LIN {X 0.029,Y -222.259,Z 1297.820,A 0.000,B 0.000,C 90.000,E1 327.533} C_DIS
LIN {X -0.001,Y -229.136,Z 1297.798,A 0.000,B 0.000,C 90.000,E1 323.703} C_DIS
LIN {X 0.049,Y -236.925,Z 1297.777,A 0.000,B 0.000,C 90.000,E1 319.908} C_DIS
LIN {X -0.024,Y -243.959,Z 1297.761,A 0.000,B 0.000,C 90.000,E1 316.944} C_DIS
LIN {X 0.067,Y -252.924,Z 1297.742,A 0.000,B 0.000,C 90.000,E1 313.623} C_DIS
LIN {X -0.154,Y -260.714,Z 1297.728,A 0.000,B 0.000,C 90.000,E1 311.148} C_DIS
LIN {X -0.101,Y -267.095,Z 1297.719,A 0.000,B 0.000,C 90.000,E1 309.358} C_DIS
LIN {X -0.026,Y -275.499,Z 1297.707,A 0.000,B 0.000,C 90.000,E1 307.237} C_DIS
LIN {X -0.075,Y -283.266,Z 1297.697,A 0.000,B 0.000,C 90.000,E1 305.518} C_DIS
LIN {X 0.052,Y -293.703,Z 1297.686,A 0.000,B 0.000,C 90.000,E1 303.452} C_DIS
LIN {X -0.037,Y -303.212,Z 1297.677,A 0.000,B 0.000,C 90.000,E1 301.799} C_DIS
LIN {X 0.071,Y -318.318,Z 1297.664,A 0.000,B 0.000,C 90.000,E1 299.489} C_DIS
LIN {X 0.040,Y -330.289,Z 1297.655,A 0.000,B 0.000,C 90.000,E1 297.897} C_DIS
LIN {X 0.050,Y -350.836,Z 1297.641,A 0.000,B 0.000,C 90.000,E1 295.412} C_DIS
LIN {X 0.152,Y -363.810,Z 1297.633,A 0.000,B 0.000,C 90.000,E1 293.898} C_DIS
LIN {X -0.055,Y -376.466,Z 1297.625,A 0.000,B 0.000,C 90.000,E1 292.461} C_DIS
LIN {X 0.202,Y -388.826,Z 1297.617,A 0.000,B 0.000,C 90.000,E1 290.972} C_DIS
LIN {X 0.126,Y -413.426,Z 1297.601,A 0.000,B 0.000,C 90.000,E1 288.181} C_DIS
LIN {X -0.186,Y -425.633,Z 1297.594,A 0.000,B 0.000,C 90.000,E1 286.858} C_DIS
LIN {X 0.004,Y -432.572,Z 1297.589,A 0.000,B 0.000,C 90.000,E1 286.024} C_DIS
LIN {X -0.170,Y -438.889,Z 1297.585,A 0.000,B 0.000,C 90.000,E1 285.245} C_DIS
LIN {X -0.194,Y -442.664,Z 1297.582,A 0.000,B 0.000,C 90.000,E1 284.717} C_DIS
LIN {X 0.140,Y -447.628,Z 1297.577,A 0.000,B 0.000,C 90.000,E1 283.883} C_DIS
LIN {X -0.016,Y -451.995,Z 1297.573,A 0.000,B 0.000,C 90.000,E1 283.119} C_DIS
LIN {X -0.140,Y -455.836,Z 1297.568,A 0.000,B 0.000,C 90.000,E1 282.355} C_DIS
LIN {X -0.055,Y -458.106,Z 1297.566,A 0.000,B 0.000,C 90.000,E1 281.827} C_DIS
LIN {X 0.044,Y -460.116,Z 1297.563,A 0.000,B 0.000,C 90.000,E1 281.299} C_DIS
LIN {X 0.063,Y -461.853,Z 1297.560,A 0.000,B 0.000,C 90.000,E1 280.782} C_DIS
LIN {X 0.181,Y -463.242,Z 1297.557,A 0.000,B 0.000,C 90.000,E1 280.254} C_DIS
LIN {X -0.150,Y -464.264,Z 1297.554,A 0.000,B 0.000,C 90.000,E1 279.782} C_DIS
LIN {X -0.095,Y -464.907,Z 1297.551,A 0.000,B 0.000,C 90.000,E1 279.265} C_DIS
LIN {X -0.030,Y -465.112,Z 1297.549,A 0.000,B 0.000,C 90.000,E1 278.746} C_DIS
LIN {X 0.108,Y -464.850,Z 1297.546,A 0.000,B 0.000,C 90.000,E1 278.219} C_DIS
LIN {X 0.179,Y -464.126,Z 1297.543,A 0.000,B 0.000,C 90.000,E1 277.701} C_DIS
LIN {X -0.210,Y -462.917,Z 1297.540,A 0.000,B 0.000,C 90.000,E1 277.239} C_DIS
LIN {X -0.142,Y -461.245,Z 1297.537,A 0.000,B 0.000,C 90.000,E1 276.720} C_DIS
LIN {X -0.081,Y -459.120,Z 1297.534,A 0.000,B 0.000,C 90.000,E1 276.201} C_DIS
LIN {X -0.030,Y -456.577,Z 1297.531,A 0.000,B 0.000,C 90.000,E1 275.682} C_DIS
LIN {X 0.001,Y -453.548,Z 1297.529,A 0.000,B 0.000,C 90.000,E1 275.163} C_DIS
LIN {X 0.013,Y -449.938,Z 1297.526,A 0.000,B 0.000,C 90.000,E1 274.645} C_DIS
LIN {X -0.028,Y -445.480,Z 1297.523,A 0.000,B 0.000,C 90.000,E1 274.131} C_DIS
LIN {X 0.194,Y -442.859,Z 1297.521,A 0.000,B 0.000,C 90.000,E1 273.841} C_DIS
LIN {X -0.088,Y -437.026,Z 1297.519,A 0.000,B 0.000,C 90.000,E1 273.383} C_DIS
LIN {X 0.058,Y -430.812,Z 1297.516,A 0.000,B 0.000,C 90.000,E1 272.922} C_DIS
LIN {X 0.169,Y -424.141,Z 1297.514,A 0.000,B 0.000,C 90.000,E1 272.522} C_DIS
LIN {X -0.134,Y -417.304,Z 1297.512,A 0.000,B 0.000,C 90.000,E1 272.236} C_DIS
LIN {X -0.049,Y -410.193,Z 1297.511,A 0.000,B 0.000,C 90.000,E1 271.949} C_DIS
LIN {X -0.028,Y -403.093,Z 1297.510,A 0.000,B 0.000,C 90.000,E1 271.718} C_DIS
LIN {X -0.139,Y -395.840,Z 1297.508,A 0.000,B 0.000,C 90.000,E1 271.547} C_DIS
LIN {X -0.014,Y -388.314,Z 1297.508,A 0.000,B 0.000,C 90.000,E1 271.375} C_DIS
LIN {X -0.082,Y -379.859,Z 1297.507,A 0.000,B 0.000,C 90.000,E1 271.260} C_DIS
LIN {X 0.025,Y -369.869,Z 1297.506,A 0.000,B 0.000,C 90.000,E1 271.146} C_DIS
LIN {X 0.116,Y -361.500,Z 1297.506,A 0.000,B 0.000,C 90.000,E1 271.088} C_DIS
LIN {X 0.020,Y -355.047,Z 1297.506,A 0.000,B 0.000,C 90.000,E1 271.088} C_DIS
LIN {X -0.014,Y -181.437,Z 1297.506,A 0.000,B 0.000,C 90.000,E1 271.088} C_DIS
LIN {X -0.077,Y -181.580,Z 1297.501,A 0.000,B 0.000,C 90.000,E1 270.229} C_DIS
LIN {X 0.092,Y -180.889,Z 1297.473,A 0.000,B 0.000,C 90.000,E1 265.122} C_DIS
LIN {X -0.026,Y -179.014,Z 1297.445,A 0.000,B 0.000,C 90.000,E1 260.095} C_DIS
LIN {X 0.069,Y -178.636,Z 1297.440,A 0.000,B 0.000,C 90.000,E1 259.218} C_DIS
LIN {X -0.033,Y -175.686,Z 1297.412,A 0.000,B 0.000,C 90.000,E1 254.157} C_DIS
LIN {X -0.022,Y -172.403,Z 1297.388,A 0.000,B 0.000,C 90.000,E1 249.880} C_DIS
LIN {X -0.005,Y -171.214,Z 1297.379,A 0.000,B 0.000,C 90.000,E1 248.156} C_DIS
LIN {X -0.029,Y -167.498,Z 1297.355,A 0.000,B 0.000,C 90.000,E1 243.845} C_DIS
LIN {X 0.053,Y -166.894,Z 1297.350,A 0.000,B 0.000,C 90.000,E1 242.948} C_DIS
LIN {X 0.043,Y -162.201,Z 1297.321,A 0.000,B 0.000,C 90.000,E1 237.709} C_DIS
LIN {X 0.011,Y -160.774,Z 1297.311,A 0.000,B 0.000,C 90.000,E1 235.960} C_DIS
LIN {X -0.018,Y -157.568,Z 1297.291,A 0.000,B 0.000,C 90.000,E1 232.431} C_DIS
LIN {X 0.017,Y -155.599,Z 1297.276,A 0.000,B 0.000,C 90.000,E1 229.747} C_DIS
LIN {X 0.067,Y -151.880,Z 1297.251,A 0.000,B 0.000,C 90.000,E1 225.243} C_DIS
LIN {X 0.081,Y -150.106,Z 1297.236,A 0.000,B 0.000,C 90.000,E1 222.528} C_DIS
LIN {X -0.003,Y -146.903,Z 1297.211,A 0.000,B 0.000,C 90.000,E1 218.016} C_DIS
LIN {X 0.017,Y -145.490,Z 1297.196,A 0.000,B 0.000,C 90.000,E1 215.264} C_DIS
LIN {X 0.017,Y -142.897,Z 1297.170,A 0.000,B 0.000,C 90.000,E1 210.669} C_DIS
LIN {X -0.052,Y -141.516,Z 1297.150,A 0.000,B 0.000,C 90.000,E1 207.001} C_DIS
LIN {X -0.009,Y -139.393,Z 1297.114,A 0.000,B 0.000,C 90.000,E1 200.482} C_DIS
LIN {X 0.042,Y -139.104,Z 1297.103,A 0.000,B 0.000,C 90.000,E1 198.598} C_DIS
LIN {X 0.034,Y -138.353,Z 1297.057,A 0.000,B 0.000,C 90.000,E1 190.197} C_DIS
LIN {X 0.027,Y -139.512,Z 1297.005,A 0.000,B 0.000,C 90.000,E1 180.859} C_DIS
LIN {X -0.032,Y -141.159,Z 1296.974,A 0.000,B 0.000,C 90.000,E1 175.298} C_DIS
LIN {X -0.061,Y -142.539,Z 1296.958,A 0.000,B 0.000,C 90.000,E1 172.527} C_DIS
LIN {X 0.006,Y -144.809,Z 1296.933,A 0.000,B 0.000,C 90.000,E1 167.881} C_DIS
LIN {X -0.006,Y -147.428,Z 1296.912,A 0.000,B 0.000,C 90.000,E1 164.212} C_DIS
LIN {X 0.022,Y -150.008,Z 1296.892,A 0.000,B 0.000,C 90.000,E1 160.550} C_DIS
LIN {X 0.030,Y -153.339,Z 1296.872,A 0.000,B 0.000,C 90.000,E1 156.922} C_DIS
LIN {X 0.011,Y -155.874,Z 1296.857,A 0.000,B 0.000,C 90.000,E1 154.229} C_DIS
LIN {X -0.022,Y -159.728,Z 1296.837,A 0.000,B 0.000,C 90.000,E1 150.667} C_DIS
LIN {X 0.044,Y -161.967,Z 1296.827,A 0.000,B 0.000,C 90.000,E1 148.869} C_DIS
LIN {X -0.071,Y -166.158,Z 1296.808,A 0.000,B 0.000,C 90.000,E1 145.388} C_DIS
LIN {X -0.076,Y -171.172,Z 1296.788,A 0.000,B 0.000,C 90.000,E1 141.904} C_DIS
LIN {X -0.042,Y -176.052,Z 1296.769,A 0.000,B 0.000,C 90.000,E1 138.447} C_DIS
LIN {X -0.047,Y -180.308,Z 1296.755,A 0.000,B 0.000,C 90.000,E1 135.891} C_DIS
LIN {X -0.076,Y -185.719,Z 1296.736,A 0.000,B 0.000,C 90.000,E1 132.528} C_DIS
LIN {X -0.024,Y -190.327,Z 1296.722,A 0.000,B 0.000,C 90.000,E1 130.011} C_DIS
LIN {X 0.023,Y -197.653,Z 1296.699,A 0.000,B 0.000,C 90.000,E1 125.884} C_DIS
LIN {X -0.040,Y -199.574,Z 1296.694,A 0.000,B 0.000,C 90.000,E1 124.945} C_DIS
LIN {X -0.098,Y -309.336,Z 1296.694,A 0.000,B 0.000,C 90.000,E1 124.945} C_DIS
LIN {X -0.078,Y -311.539,Z 1296.694,A 0.000,B 0.000,C 90.000,E1 124.898} C_DIS
LIN {X 0.053,Y -316.988,Z 1296.692,A 0.000,B 0.000,C 90.000,E1 124.565} C_DIS
LIN {X -0.076,Y -319.924,Z 1296.690,A 0.000,B 0.000,C 90.000,E1 124.278} C_DIS
LIN {X -0.103,Y -321.931,Z 1296.689,A 0.000,B 0.000,C 90.000,E1 123.992} C_DIS
LIN {X -0.130,Y -323.499,Z 1296.687,A 0.000,B 0.000,C 90.000,E1 123.706} C_DIS
LIN {X -0.043,Y -324.854,Z 1296.685,A 0.000,B 0.000,C 90.000,E1 123.372} C_DIS
LIN {X 0.054,Y -336.500,Z 1296.668,A 0.000,B 0.000,C 90.000,E1 120.207} C_DIS
LIN {X 0.008,Y -348.385,Z 1296.652,A 0.000,B 0.000,C 90.000,E1 117.436} C_DIS
LIN {X -0.025,Y -361.721,Z 1296.637,A 0.000,B 0.000,C 90.000,E1 114.719} C_DIS
LIN {X 0.081,Y -374.891,Z 1296.624,A 0.000,B 0.000,C 90.000,E1 112.333} C_DIS
LIN {X 0.233,Y -389.393,Z 1296.611,A 0.000,B 0.000,C 90.000,E1 109.993} C_DIS
LIN {X -0.019,Y -405.329,Z 1296.599,A 0.000,B 0.000,C 90.000,E1 107.764} C_DIS
LIN {X 0.002,Y -422.809,Z 1296.586,A 0.000,B 0.000,C 90.000,E1 105.552} C_DIS
LIN {X -0.060,Y -441.930,Z 1296.574,A 0.000,B 0.000,C 90.000,E1 103.411} C_DIS
LIN {X -0.233,Y -462.017,Z 1296.563,A 0.000,B 0.000,C 90.000,E1 101.422} C_DIS
LIN {X -0.198,Y -477.377,Z 1296.556,A 0.000,B 0.000,C 90.000,E1 100.018} C_DIS
LIN {X -0.117,Y -479.361,Z 1296.554,A 0.000,B 0.000,C 90.000,E1 99.782} C_DIS
LIN {X 0.148,Y -481.022,Z 1296.553,A 0.000,B 0.000,C 90.000,E1 99.500} C_DIS
LIN {X 0.022,Y -482.268,Z 1296.552,A 0.000,B 0.000,C 90.000,E1 99.265} C_DIS
LIN {X 0.188,Y -483.795,Z 1296.549,A 0.000,B 0.000,C 90.000,E1 98.746} C_DIS
LIN {X -0.046,Y -484.267,Z 1296.546,A 0.000,B 0.000,C 90.000,E1 98.276} C_DIS
LIN {X 0.136,Y -483.763,Z 1296.543,A 0.000,B 0.000,C 90.000,E1 97.757} C_DIS
LIN {X -0.156,Y -482.204,Z 1296.540,A 0.000,B 0.000,C 90.000,E1 97.296} C_DIS
LIN {X 0.145,Y -480.944,Z 1296.539,A 0.000,B 0.000,C 90.000,E1 97.011} C_DIS
LIN {X 0.028,Y -479.266,Z 1296.538,A 0.000,B 0.000,C 90.000,E1 96.777} C_DIS
LIN {X -0.011,Y -467.993,Z 1296.529,A 0.000,B 0.000,C 90.000,E1 95.277} C_DIS
LIN {X 0.186,Y -454.112,Z 1296.518,A 0.000,B 0.000,C 90.000,E1 93.212} C_DIS
LIN {X -0.019,Y -437.481,Z 1296.504,A 0.000,B 0.000,C 90.000,E1 90.630} C_DIS
LIN {X -0.017,Y -419.690,Z 1296.486,A 0.000,B 0.000,C 90.000,E1 87.421} C_DIS
LIN {X -0.061,Y -408.148,Z 1296.474,A 0.000,B 0.000,C 90.000,E1 85.241} C_DIS
LIN {X 0.054,Y -397.889,Z 1296.463,A 0.000,B 0.000,C 90.000,E1 83.280} C_DIS
LIN {X -0.039,Y -387.490,Z 1296.452,A 0.000,B 0.000,C 90.000,E1 81.319} C_DIS
LIN {X 0.115,Y -378.224,Z 1296.442,A 0.000,B 0.000,C 90.000,E1 79.577} C_DIS
LIN {X -0.197,Y -370.312,Z 1296.434,A 0.000,B 0.000,C 90.000,E1 78.173} C_DIS
LIN {X 0.150,Y -360.564,Z 1296.424,A 0.000,B 0.000,C 90.000,E1 76.353} C_DIS
LIN {X -0.012,Y -348.993,Z 1296.413,A 0.000,B 0.000,C 90.000,E1 74.283} C_DIS
LIN {X 0.100,Y -337.395,Z 1296.401,A 0.000,B 0.000,C 90.000,E1 72.127} C_DIS
LIN {X 0.029,Y -324.338,Z 1296.387,A 0.000,B 0.000,C 90.000,E1 69.645} C_DIS
LIN {X -0.165,Y -309.001,Z 1296.369,A 0.000,B 0.000,C 90.000,E1 66.485} C_DIS
LIN {X -0.029,Y -296.366,Z 1296.353,A 0.000,B 0.000,C 90.000,E1 63.512} C_DIS
LIN {X -0.050,Y -288.933,Z 1296.342,A 0.000,B 0.000,C 90.000,E1 61.513} C_DIS
LIN {X 0.010,Y -280.189,Z 1296.327,A 0.000,B 0.000,C 90.000,E1 58.791} C_DIS
LIN {X 0.034,Y -270.342,Z 1296.307,A 0.000,B 0.000,C 90.000,E1 55.341} C_DIS
LIN {X 0.075,Y -261.296,Z 1296.288,A 0.000,B 0.000,C 90.000,E1 51.823} C_DIS
LIN {X -0.107,Y -254.319,Z 1296.272,A 0.000,B 0.000,C 90.000,E1 49.013} C_DIS
LIN {X -0.150,Y -247.597,Z 1296.256,A 0.000,B 0.000,C 90.000,E1 46.134} C_DIS
LIN {X -0.057,Y -239.525,Z 1296.236,A 0.000,B 0.000,C 90.000,E1 42.447} C_DIS
LIN {X 0.013,Y -232.214,Z 1296.215,A 0.000,B 0.000,C 90.000,E1 38.705} C_DIS
LIN {X -0.069,Y -225.785,Z 1296.194,A 0.000,B 0.000,C 90.000,E1 34.945} C_DIS
LIN {X 0.062,Y -220.215,Z 1296.173,A 0.000,B 0.000,C 90.000,E1 31.082} C_DIS
LIN {X 0.070,Y -215.505,Z 1296.151,A 0.000,B 0.000,C 90.000,E1 27.206} C_DIS
LIN {X 0.045,Y -210.493,Z 1296.125,A 0.000,B 0.000,C 90.000,E1 22.514} C_DIS
LIN {X -0.087,Y -206.837,Z 1296.103,A 0.000,B 0.000,C 90.000,E1 18.598} C_DIS
LIN {X 0.065,Y -203.016,Z 1296.077,A 0.000,B 0.000,C 90.000,E1 13.772} C_DIS
LIN {X -0.013,Y -200.039,Z 1296.050,A 0.000,B 0.000,C 90.000,E1 8.973} C_DIS
LIN {X -0.086,Y -197.636,Z 1296.014,A 0.000,B 0.000,C 90.000,E1 2.522} C_DIS
LIN {X -0.072,Y -197.833,Z 1295.961,A 0.000,B 0.000,C 90.000,E1 353.053} C_DIS
LIN {X 0.065,Y -200.799,Z 1295.925,A 0.000,B 0.000,C 90.000,E1 346.533} C_DIS
LIN {X 0.052,Y -204.515,Z 1295.898,A 0.000,B 0.000,C 90.000,E1 341.710} C_DIS
LIN {X 0.064,Y -209.284,Z 1295.872,A 0.000,B 0.000,C 90.000,E1 336.922} C_DIS
LIN {X -0.032,Y -214.177,Z 1295.850,A 0.000,B 0.000,C 90.000,E1 332.999} C_DIS
LIN {X 0.034,Y -219.832,Z 1295.828,A 0.000,B 0.000,C 90.000,E1 329.076} C_DIS
LIN {X -0.010,Y -226.312,Z 1295.807,A 0.000,B 0.000,C 90.000,E1 325.229} C_DIS
LIN {X 0.039,Y -233.704,Z 1295.786,A 0.000,B 0.000,C 90.000,E1 321.412} C_DIS
LIN {X -0.003,Y -242.146,Z 1295.765,A 0.000,B 0.000,C 90.000,E1 317.676} C_DIS
LIN {X -0.137,Y -251.903,Z 1295.744,A 0.000,B 0.000,C 90.000,E1 314.028} C_DIS
LIN {X -0.014,Y -259.554,Z 1295.730,A 0.000,B 0.000,C 90.000,E1 311.472} C_DIS
LIN {X -0.012,Y -265.764,Z 1295.720,A 0.000,B 0.000,C 90.000,E1 309.688} C_DIS
LIN {X -0.046,Y -275.505,Z 1295.707,A 0.000,B 0.000,C 90.000,E1 307.237} C_DIS
LIN {X -0.096,Y -283.273,Z 1295.697,A 0.000,B 0.000,C 90.000,E1 305.518} C_DIS
LIN {X 0.031,Y -293.693,Z 1295.686,A 0.000,B 0.000,C 90.000,E1 303.452} C_DIS
LIN {X -0.059,Y -303.226,Z 1295.677,A 0.000,B 0.000,C 90.000,E1 301.799} C_DIS
LIN {X 0.148,Y -316.069,Z 1295.666,A 0.000,B 0.000,C 90.000,E1 299.795} C_DIS
LIN {X -0.083,Y -327.805,Z 1295.657,A 0.000,B 0.000,C 90.000,E1 298.231} C_DIS
LIN {X 0.152,Y -347.974,Z 1295.643,A 0.000,B 0.000,C 90.000,E1 295.720} C_DIS
LIN {X -0.025,Y -363.532,Z 1295.633,A 0.000,B 0.000,C 90.000,E1 293.951} C_DIS
LIN {X -0.167,Y -376.094,Z 1295.625,A 0.000,B 0.000,C 90.000,E1 292.514} C_DIS
LIN {X -0.047,Y -388.446,Z 1295.617,A 0.000,B 0.000,C 90.000,E1 291.046} C_DIS
LIN {X 0.141,Y -412.885,Z 1295.601,A 0.000,B 0.000,C 90.000,E1 288.236} C_DIS
LIN {X -0.187,Y -425.163,Z 1295.594,A 0.000,B 0.000,C 90.000,E1 286.913} C_DIS
LIN {X -0.021,Y -432.154,Z 1295.589,A 0.000,B 0.000,C 90.000,E1 286.079} C_DIS
LIN {X 0.222,Y -438.543,Z 1295.585,A 0.000,B 0.000,C 90.000,E1 285.245} C_DIS
LIN {X 0.199,Y -442.337,Z 1295.582,A 0.000,B 0.000,C 90.000,E1 284.717} C_DIS
LIN {X -0.007,Y -447.446,Z 1295.578,A 0.000,B 0.000,C 90.000,E1 283.953} C_DIS
LIN {X -0.060,Y -451.877,Z 1295.573,A 0.000,B 0.000,C 90.000,E1 283.175} C_DIS
LIN {X -0.187,Y -455.766,Z 1295.569,A 0.000,B 0.000,C 90.000,E1 282.411} C_DIS
LIN {X -0.103,Y -458.045,Z 1295.566,A 0.000,B 0.000,C 90.000,E1 281.883} C_DIS
LIN {X -0.096,Y -460.076,Z 1295.563,A 0.000,B 0.000,C 90.000,E1 281.366} C_DIS
LIN {X 0.012,Y -461.868,Z 1295.560,A 0.000,B 0.000,C 90.000,E1 280.838} C_DIS
LIN {X 0.130,Y -463.299,Z 1295.557,A 0.000,B 0.000,C 90.000,E1 280.310} C_DIS
LIN {X 0.177,Y -464.326,Z 1295.555,A 0.000,B 0.000,C 90.000,E1 279.792} C_DIS
LIN {X -0.148,Y -465.047,Z 1295.552,A 0.000,B 0.000,C 90.000,E1 279.321} C_DIS
LIN {X -0.084,Y -465.307,Z 1295.549,A 0.000,B 0.000,C 90.000,E1 278.803} C_DIS
LIN {X 0.055,Y -465.123,Z 1295.546,A 0.000,B 0.000,C 90.000,E1 278.276} C_DIS
LIN {X 0.126,Y -464.444,Z 1295.543,A 0.000,B 0.000,C 90.000,E1 277.757} C_DIS
LIN {X 0.198,Y -463.340,Z 1295.540,A 0.000,B 0.000,C 90.000,E1 277.239} C_DIS
LIN {X -0.193,Y -461.749,Z 1295.537,A 0.000,B 0.000,C 90.000,E1 276.777} C_DIS
LIN {X -0.129,Y -459.662,Z 1295.535,A 0.000,B 0.000,C 90.000,E1 276.258} C_DIS
LIN {X 0.147,Y -455.800,Z 1295.530,A 0.000,B 0.000,C 90.000,E1 275.454} C_DIS
LIN {X 0.173,Y -452.631,Z 1295.528,A 0.000,B 0.000,C 90.000,E1 274.935} C_DIS
LIN {X 0.180,Y -448.776,Z 1295.525,A 0.000,B 0.000,C 90.000,E1 274.416} C_DIS
LIN {X 0.164,Y -444.031,Z 1295.522,A 0.000,B 0.000,C 90.000,E1 273.898} C_DIS
LIN {X -0.169,Y -438.312,Z 1295.519,A 0.000,B 0.000,C 90.000,E1 273.440} C_DIS
LIN {X -0.094,Y -432.145,Z 1295.516,A 0.000,B 0.000,C 90.000,E1 272.980} C_DIS
LIN {X -0.052,Y -425.578,Z 1295.514,A 0.000,B 0.000,C 90.000,E1 272.579} C_DIS
LIN {X 0.014,Y -418.754,Z 1295.512,A 0.000,B 0.000,C 90.000,E1 272.236} C_DIS
LIN {X 0.088,Y -411.753,Z 1295.511,A 0.000,B 0.000,C 90.000,E1 271.949} C_DIS
LIN {X 0.068,Y -404.712,Z 1295.510,A 0.000,B 0.000,C 90.000,E1 271.718} C_DIS
LIN {X -0.109,Y -397.480,Z 1295.509,A 0.000,B 0.000,C 90.000,E1 271.547} C_DIS
LIN {X -0.121,Y -385.844,Z 1295.507,A 0.000,B 0.000,C 90.000,E1 271.318} C_DIS
LIN {X -0.140,Y -376.720,Z 1295.507,A 0.000,B 0.000,C 90.000,E1 271.203} C_DIS
LIN {X 0.023,Y -364.736,Z 1295.506,A 0.000,B 0.000,C 90.000,E1 271.088} C_DIS
LIN {X -0.128,Y -357.474,Z 1295.506,A 0.000,B 0.000,C 90.000,E1 271.088} C_DIS
LIN {X -0.090,Y -181.442,Z 1295.506,A 0.000,B 0.000,C 90.000,E1 271.088} C_DIS
LIN {X 0.045,Y -181.579,Z 1295.501,A 0.000,B 0.000,C 90.000,E1 270.172} C_DIS
LIN {X 0.033,Y -180.887,Z 1295.473,A 0.000,B 0.000,C 90.000,E1 265.122} C_DIS
LIN {X -0.084,Y -179.009,Z 1295.445,A 0.000,B 0.000,C 90.000,E1 260.095} C_DIS
LIN {X 0.011,Y -178.622,Z 1295.440,A 0.000,B 0.000,C 90.000,E1 259.218} C_DIS
LIN {X -0.090,Y -175.674,Z 1295.412,A 0.000,B 0.000,C 90.000,E1 254.157} C_DIS
LIN {X -0.078,Y -172.390,Z 1295.388,A 0.000,B 0.000,C 90.000,E1 249.880} C_DIS
LIN {X -0.061,Y -171.194,Z 1295.379,A 0.000,B 0.000,C 90.000,E1 248.156} C_DIS
LIN {X -0.011,Y -167.484,Z 1295.354,A 0.000,B 0.000,C 90.000,E1 243.819} C_DIS
LIN {X -0.003,Y -166.881,Z 1295.350,A 0.000,B 0.000,C 90.000,E1 242.948} C_DIS
LIN {X -0.011,Y -162.186,Z 1295.321,A 0.000,B 0.000,C 90.000,E1 237.709} C_DIS
LIN {X 0.046,Y -160.755,Z 1295.311,A 0.000,B 0.000,C 90.000,E1 235.928} C_DIS
LIN {X 0.025,Y -157.552,Z 1295.291,A 0.000,B 0.000,C 90.000,E1 232.396} C_DIS
LIN {X -0.037,Y -155.581,Z 1295.276,A 0.000,B 0.000,C 90.000,E1 229.747} C_DIS
LIN {X 0.014,Y -151.866,Z 1295.251,A 0.000,B 0.000,C 90.000,E1 225.243} C_DIS
LIN {X 0.028,Y -150.090,Z 1295.236,A 0.000,B 0.000,C 90.000,E1 222.528} C_DIS
LIN {X -0.054,Y -146.891,Z 1295.211,A 0.000,B 0.000,C 90.000,E1 218.016} C_DIS
LIN {X 0.050,Y -145.477,Z 1295.196,A 0.000,B 0.000,C 90.000,E1 215.231} C_DIS
LIN {X -0.033,Y -142.888,Z 1295.170,A 0.000,B 0.000,C 90.000,E1 210.669} C_DIS
LIN {X 0.024,Y -141.507,Z 1295.150,A 0.000,B 0.000,C 90.000,E1 206.950} C_DIS
LIN {X -0.058,Y -139.391,Z 1295.114,A 0.000,B 0.000,C 90.000,E1 200.482} C_DIS
LIN {X -0.007,Y -139.098,Z 1295.103,A 0.000,B 0.000,C 90.000,E1 198.598} C_DIS
LIN {X -0.015,Y -138.354,Z 1295.057,A 0.000,B 0.000,C 90.000,E1 190.197} C_DIS
LIN {X -0.022,Y -139.515,Z 1295.005,A 0.000,B 0.000,C 90.000,E1 180.859} C_DIS
LIN {X 0.058,Y -141.167,Z 1294.974,A 0.000,B 0.000,C 90.000,E1 175.241} C_DIS
LIN {X 0.030,Y -142.546,Z 1294.958,A 0.000,B 0.000,C 90.000,E1 172.470} C_DIS
LIN {X -0.044,Y -144.822,Z 1294.933,A 0.000,B 0.000,C 90.000,E1 167.881} C_DIS
LIN {X -0.058,Y -147.443,Z 1294.912,A 0.000,B 0.000,C 90.000,E1 164.212} C_DIS
LIN {X -0.029,Y -150.024,Z 1294.892,A 0.000,B 0.000,C 90.000,E1 160.550} C_DIS
LIN {X -0.023,Y -153.359,Z 1294.872,A 0.000,B 0.000,C 90.000,E1 156.922} C_DIS
LIN {X 0.025,Y -155.893,Z 1294.857,A 0.000,B 0.000,C 90.000,E1 154.204} C_DIS
LIN {X -0.077,Y -159.751,Z 1294.837,A 0.000,B 0.000,C 90.000,E1 150.667} C_DIS
LIN {X -0.011,Y -161.991,Z 1294.827,A 0.000,B 0.000,C 90.000,E1 148.869} C_DIS
LIN {X 0.009,Y -166.184,Z 1294.807,A 0.000,B 0.000,C 90.000,E1 145.341} C_DIS
LIN {X 0.107,Y -171.198,Z 1294.788,A 0.000,B 0.000,C 90.000,E1 141.823} C_DIS
LIN {X 0.032,Y -176.082,Z 1294.769,A 0.000,B 0.000,C 90.000,E1 138.405} C_DIS
LIN {X -0.107,Y -180.342,Z 1294.755,A 0.000,B 0.000,C 90.000,E1 135.891} C_DIS
LIN {X 0.002,Y -185.751,Z 1294.736,A 0.000,B 0.000,C 90.000,E1 132.486} C_DIS
LIN {X -0.085,Y -190.363,Z 1294.722,A 0.000,B 0.000,C 90.000,E1 130.011} C_DIS
LIN {X -0.039,Y -197.688,Z 1294.699,A 0.000,B 0.000,C 90.000,E1 125.884} C_DIS
LIN {X 0.062,Y -199.611,Z 1294.694,A 0.000,B 0.000,C 90.000,E1 124.898} C_DIS
LIN {X 0.060,Y -309.034,Z 1294.694,A 0.000,B 0.000,C 90.000,E1 124.898} C_DIS
LIN {X -0.175,Y -311.492,Z 1294.694,A 0.000,B 0.000,C 90.000,E1 124.898} C_DIS
LIN {X 0.134,Y -317.004,Z 1294.692,A 0.000,B 0.000,C 90.000,E1 124.532} C_DIS
LIN {X 0.005,Y -319.951,Z 1294.690,A 0.000,B 0.000,C 90.000,E1 124.246} C_DIS
LIN {X -0.199,Y -321.959,Z 1294.689,A 0.000,B 0.000,C 90.000,E1 123.992} C_DIS
LIN {X 0.047,Y -323.528,Z 1294.687,A 0.000,B 0.000,C 90.000,E1 123.658} C_DIS
LIN {X -0.135,Y -324.887,Z 1294.685,A 0.000,B 0.000,C 90.000,E1 123.372} C_DIS
LIN {X -0.040,Y -336.543,Z 1294.668,A 0.000,B 0.000,C 90.000,E1 120.207} C_DIS
LIN {X -0.088,Y -348.436,Z 1294.652,A 0.000,B 0.000,C 90.000,E1 117.436} C_DIS
LIN {X 0.028,Y -361.780,Z 1294.637,A 0.000,B 0.000,C 90.000,E1 114.695} C_DIS
LIN {X -0.018,Y -374.957,Z 1294.624,A 0.000,B 0.000,C 90.000,E1 112.333} C_DIS
LIN {X 0.131,Y -389.468,Z 1294.611,A 0.000,B 0.000,C 90.000,E1 109.993} C_DIS
LIN {X -0.123,Y -405.413,Z 1294.599,A 0.000,B 0.000,C 90.000,E1 107.764} C_DIS
LIN {X -0.105,Y -422.904,Z 1294.586,A 0.000,B 0.000,C 90.000,E1 105.552} C_DIS
LIN {X -0.168,Y -442.035,Z 1294.574,A 0.000,B 0.000,C 90.000,E1 103.411} C_DIS
LIN {X 0.115,Y -462.125,Z 1294.563,A 0.000,B 0.000,C 90.000,E1 101.366} C_DIS
LIN {X 0.170,Y -477.455,Z 1294.555,A 0.000,B 0.000,C 90.000,E1 99.962} C_DIS
LIN {X 0.253,Y -479.387,Z 1294.554,A 0.000,B 0.000,C 90.000,E1 99.726} C_DIS
LIN {X 0.046,Y -481.008,Z 1294.553,A 0.000,B 0.000,C 90.000,E1 99.500} C_DIS
LIN {X -0.081,Y -482.223,Z 1294.551,A 0.000,B 0.000,C 90.000,E1 99.265} C_DIS
LIN {X 0.084,Y -483.703,Z 1294.549,A 0.000,B 0.000,C 90.000,E1 98.746} C_DIS
LIN {X -0.149,Y -484.134,Z 1294.546,A 0.000,B 0.000,C 90.000,E1 98.276} C_DIS
LIN {X 0.033,Y -483.589,Z 1294.543,A 0.000,B 0.000,C 90.000,E1 97.757} C_DIS
LIN {X 0.218,Y -481.982,Z 1294.540,A 0.000,B 0.000,C 90.000,E1 97.239} C_DIS
LIN {X 0.100,Y -480.692,Z 1294.539,A 0.000,B 0.000,C 90.000,E1 97.004} C_DIS
LIN {X -0.203,Y -477.018,Z 1294.536,A 0.000,B 0.000,C 90.000,E1 96.543} C_DIS
LIN {X 0.144,Y -465.938,Z 1294.528,A 0.000,B 0.000,C 90.000,E1 94.992} C_DIS
LIN {X 0.077,Y -453.816,Z 1294.518,A 0.000,B 0.000,C 90.000,E1 93.212} C_DIS
LIN {X -0.133,Y -437.196,Z 1294.503,A 0.000,B 0.000,C 90.000,E1 90.630} C_DIS
LIN {X -0.136,Y -419.389,Z 1294.486,A 0.000,B 0.000,C 90.000,E1 87.421} C_DIS
LIN {X -0.184,Y -407.845,Z 1294.473,A 0.000,B 0.000,C 90.000,E1 85.241} C_DIS
LIN {X -0.072,Y -397.604,Z 1294.463,A 0.000,B 0.000,C 90.000,E1 83.280} C_DIS
LIN {X -0.110,Y -387.204,Z 1294.452,A 0.000,B 0.000,C 90.000,E1 81.310} C_DIS
LIN {X 0.053,Y -377.948,Z 1294.442,A 0.000,B 0.000,C 90.000,E1 79.567} C_DIS
LIN {X 0.034,Y -370.056,Z 1294.434,A 0.000,B 0.000,C 90.000,E1 78.117} C_DIS
LIN {X 0.017,Y -360.293,Z 1294.424,A 0.000,B 0.000,C 90.000,E1 76.353} C_DIS
LIN {X -0.083,Y -350.372,Z 1294.414,A 0.000,B 0.000,C 90.000,E1 74.574} C_DIS
LIN {X 0.071,Y -338.788,Z 1294.402,A 0.000,B 0.000,C 90.000,E1 72.417} C_DIS
LIN {X 0.073,Y -327.303,Z 1294.390,A 0.000,B 0.000,C 90.000,E1 70.242} C_DIS
LIN {X -0.071,Y -313.271,Z 1294.374,A 0.000,B 0.000,C 90.000,E1 67.411} C_DIS
LIN {X -0.058,Y -298.865,Z 1294.356,A 0.000,B 0.000,C 90.000,E1 64.152} C_DIS
LIN {X -0.031,Y -291.151,Z 1294.345,A 0.000,B 0.000,C 90.000,E1 62.153} C_DIS
LIN {X -0.064,Y -282.123,Z 1294.330,A 0.000,B 0.000,C 90.000,E1 59.459} C_DIS
LIN {X 0.028,Y -272.109,Z 1294.311,A 0.000,B 0.000,C 90.000,E1 56.008} C_DIS
LIN {X 0.025,Y -262.903,Z 1294.292,A 0.000,B 0.000,C 90.000,E1 52.512} C_DIS
LIN {X 0.042,Y -255.883,Z 1294.276,A 0.000,B 0.000,C 90.000,E1 49.666} C_DIS
LIN {X 0.054,Y -249.068,Z 1294.260,A 0.000,B 0.000,C 90.000,E1 46.782} C_DIS
LIN {X 0.039,Y -242.495,Z 1294.244,A 0.000,B 0.000,C 90.000,E1 43.866} C_DIS
LIN {X -0.005,Y -234.845,Z 1294.223,A 0.000,B 0.000,C 90.000,E1 40.172} C_DIS
LIN {X -0.050,Y -228.066,Z 1294.202,A 0.000,B 0.000,C 90.000,E1 36.423} C_DIS
LIN {X -0.103,Y -222.120,Z 1294.181,A 0.000,B 0.000,C 90.000,E1 32.625} C_DIS
LIN {X -0.010,Y -217.081,Z 1294.160,A 0.000,B 0.000,C 90.000,E1 28.743} C_DIS
LIN {X -0.021,Y -212.599,Z 1294.138,A 0.000,B 0.000,C 90.000,E1 24.847} C_DIS
LIN {X -0.043,Y -208.655,Z 1294.116,A 0.000,B 0.000,C 90.000,E1 20.918} C_DIS
LIN {X 0.089,Y -205.134,Z 1294.094,A 0.000,B 0.000,C 90.000,E1 16.913} C_DIS
LIN {X 0.066,Y -201.566,Z 1294.067,A 0.000,B 0.000,C 90.000,E1 12.119} C_DIS
LIN {X 0.005,Y -198.296,Z 1294.032,A 0.000,B 0.000,C 90.000,E1 5.682} C_DIS
LIN {X -0.073,Y -196.913,Z 1293.993,A 0.000,B 0.000,C 90.000,E1 358.740} C_DIS
LIN {X -0.071,Y -198.905,Z 1293.943,A 0.000,B 0.000,C 90.000,E1 349.803} C_DIS
LIN {X -0.103,Y -202.480,Z 1293.912,A 0.000,B 0.000,C 90.000,E1 344.157} C_DIS
LIN {X -0.061,Y -206.749,Z 1293.885,A 0.000,B 0.000,C 90.000,E1 339.337} C_DIS
LIN {X -0.030,Y -211.189,Z 1293.863,A 0.000,B 0.000,C 90.000,E1 335.357} C_DIS
LIN {X -0.070,Y -216.350,Z 1293.841,A 0.000,B 0.000,C 90.000,E1 331.435} C_DIS
LIN {X -0.015,Y -222.349,Z 1293.820,A 0.000,B 0.000,C 90.000,E1 327.533} C_DIS
LIN {X -0.045,Y -229.212,Z 1293.798,A 0.000,B 0.000,C 90.000,E1 323.703} C_DIS
LIN {X 0.008,Y -237.028,Z 1293.777,A 0.000,B 0.000,C 90.000,E1 319.908} C_DIS
LIN {X -0.065,Y -244.039,Z 1293.761,A 0.000,B 0.000,C 90.000,E1 316.944} C_DIS
LIN {X 0.032,Y -253.994,Z 1293.740,A 0.000,B 0.000,C 90.000,E1 313.257} C_DIS
LIN {X 0.013,Y -261.968,Z 1293.726,A 0.000,B 0.000,C 90.000,E1 310.744} C_DIS
LIN {X -0.016,Y -269.803,Z 1293.715,A 0.000,B 0.000,C 90.000,E1 308.624} C_DIS
LIN {X 0.114,Y -278.530,Z 1293.703,A 0.000,B 0.000,C 90.000,E1 306.503} C_DIS
LIN {X -0.052,Y -286.632,Z 1293.693,A 0.000,B 0.000,C 90.000,E1 304.818} C_DIS
LIN {X 0.153,Y -295.555,Z 1293.684,A 0.000,B 0.000,C 90.000,E1 303.086} C_DIS
LIN {X -0.076,Y -305.269,Z 1293.675,A 0.000,B 0.000,C 90.000,E1 301.465} C_DIS
LIN {X 0.115,Y -316.062,Z 1293.666,A 0.000,B 0.000,C 90.000,E1 299.795} C_DIS
LIN {X -0.018,Y -330.278,Z 1293.655,A 0.000,B 0.000,C 90.000,E1 297.897} C_DIS
LIN {X 0.114,Y -350.589,Z 1293.641,A 0.000,B 0.000,C 90.000,E1 295.412} C_DIS
LIN {X -0.061,Y -363.495,Z 1293.633,A 0.000,B 0.000,C 90.000,E1 293.951} C_DIS
LIN {X 0.136,Y -376.079,Z 1293.625,A 0.000,B 0.000,C 90.000,E1 292.461} C_DIS
LIN {X -0.066,Y -388.409,Z 1293.617,A 0.000,B 0.000,C 90.000,E1 291.046} C_DIS
LIN {X 0.106,Y -412.909,Z 1293.601,A 0.000,B 0.000,C 90.000,E1 288.236} C_DIS
LIN {X 0.193,Y -425.192,Z 1293.594,A 0.000,B 0.000,C 90.000,E1 286.858} C_DIS
LIN {X -0.048,Y -432.183,Z 1293.589,A 0.000,B 0.000,C 90.000,E1 286.079} C_DIS
LIN {X 0.195,Y -438.602,Z 1293.585,A 0.000,B 0.000,C 90.000,E1 285.245} C_DIS
LIN {X -0.046,Y -444.222,Z 1293.580,A 0.000,B 0.000,C 90.000,E1 284.481} C_DIS
LIN {X -0.126,Y -449.089,Z 1293.576,A 0.000,B 0.000,C 90.000,E1 283.703} C_DIS
LIN {X 0.162,Y -453.362,Z 1293.572,A 0.000,B 0.000,C 90.000,E1 282.883} C_DIS
LIN {X 0.054,Y -457.113,Z 1293.567,A 0.000,B 0.000,C 90.000,E1 282.119} C_DIS
LIN {X -0.118,Y -460.269,Z 1293.563,A 0.000,B 0.000,C 90.000,E1 281.366} C_DIS
LIN {X -0.004,Y -462.035,Z 1293.560,A 0.000,B 0.000,C 90.000,E1 280.838} C_DIS
LIN {X 0.115,Y -463.443,Z 1293.557,A 0.000,B 0.000,C 90.000,E1 280.310} C_DIS
LIN {X 0.162,Y -464.503,Z 1293.555,A 0.000,B 0.000,C 90.000,E1 279.792} C_DIS
LIN {X -0.160,Y -465.216,Z 1293.552,A 0.000,B 0.000,C 90.000,E1 279.321} C_DIS
LIN {X -0.096,Y -465.482,Z 1293.549,A 0.000,B 0.000,C 90.000,E1 278.803} C_DIS
LIN {X 0.044,Y -465.332,Z 1293.546,A 0.000,B 0.000,C 90.000,E1 278.276} C_DIS
LIN {X 0.116,Y -464.694,Z 1293.543,A 0.000,B 0.000,C 90.000,E1 277.757} C_DIS
LIN {X 0.189,Y -463.593,Z 1293.540,A 0.000,B 0.000,C 90.000,E1 277.239} C_DIS
LIN {X -0.200,Y -462.013,Z 1293.537,A 0.000,B 0.000,C 90.000,E1 276.777} C_DIS
LIN {X 0.145,Y -458.758,Z 1293.533,A 0.000,B 0.000,C 90.000,E1 275.967} C_DIS
LIN {X 0.144,Y -456.112,Z 1293.530,A 0.000,B 0.000,C 90.000,E1 275.454} C_DIS
LIN {X 0.172,Y -453.039,Z 1293.528,A 0.000,B 0.000,C 90.000,E1 274.935} C_DIS
LIN {X 0.181,Y -449.231,Z 1293.525,A 0.000,B 0.000,C 90.000,E1 274.416} C_DIS
LIN {X 0.168,Y -444.592,Z 1293.522,A 0.000,B 0.000,C 90.000,E1 273.898} C_DIS
LIN {X -0.197,Y -438.946,Z 1293.519,A 0.000,B 0.000,C 90.000,E1 273.440} C_DIS
LIN {X -0.168,Y -432.747,Z 1293.516,A 0.000,B 0.000,C 90.000,E1 272.980} C_DIS
LIN {X -0.151,Y -426.164,Z 1293.514,A 0.000,B 0.000,C 90.000,E1 272.579} C_DIS
LIN {X -0.109,Y -419.247,Z 1293.512,A 0.000,B 0.000,C 90.000,E1 272.236} C_DIS
LIN {X -0.067,Y -412.275,Z 1293.511,A 0.000,B 0.000,C 90.000,E1 271.949} C_DIS
LIN {X -0.093,Y -405.137,Z 1293.510,A 0.000,B 0.000,C 90.000,E1 271.718} C_DIS
LIN {X 0.124,Y -397.841,Z 1293.508,A 0.000,B 0.000,C 90.000,E1 271.489} C_DIS
LIN {X 0.187,Y -390.208,Z 1293.507,A 0.000,B 0.000,C 90.000,E1 271.318} C_DIS
LIN {X 0.083,Y -382.099,Z 1293.507,A 0.000,B 0.000,C 90.000,E1 271.203} C_DIS
LIN {X 0.000,Y -368.929,Z 1293.506,A 0.000,B 0.000,C 90.000,E1 271.088} C_DIS
LIN {X 0.062,Y -357.442,Z 1293.506,A 0.000,B 0.000,C 90.000,E1 271.031} C_DIS
LIN {X 0.005,Y -181.448,Z 1293.506,A 0.000,B 0.000,C 90.000,E1 271.031} C_DIS
LIN {X -0.043,Y -181.578,Z 1293.501,A 0.000,B 0.000,C 90.000,E1 270.172} C_DIS
LIN {X -0.054,Y -180.883,Z 1293.473,A 0.000,B 0.000,C 90.000,E1 265.122} C_DIS
LIN {X 0.005,Y -179.003,Z 1293.445,A 0.000,B 0.000,C 90.000,E1 260.038} C_DIS
LIN {X -0.076,Y -178.602,Z 1293.440,A 0.000,B 0.000,C 90.000,E1 259.218} C_DIS
LIN {X -0.008,Y -175.654,Z 1293.412,A 0.000,B 0.000,C 90.000,E1 254.102} C_DIS
LIN {X -0.002,Y -172.373,Z 1293.388,A 0.000,B 0.000,C 90.000,E1 249.826} C_DIS
LIN {X 0.012,Y -171.166,Z 1293.378,A 0.000,B 0.000,C 90.000,E1 248.103} C_DIS
LIN {X 0.056,Y -167.464,Z 1293.354,A 0.000,B 0.000,C 90.000,E1 243.768} C_DIS
LIN {X -0.010,Y -166.860,Z 1293.349,A 0.000,B 0.000,C 90.000,E1 242.922} C_DIS
LIN {X 0.044,Y -162.164,Z 1293.320,A 0.000,B 0.000,C 90.000,E1 237.661} C_DIS
LIN {X -0.036,Y -160.724,Z 1293.311,A 0.000,B 0.000,C 90.000,E1 235.928} C_DIS
LIN {X -0.057,Y -157.529,Z 1293.291,A 0.000,B 0.000,C 90.000,E1 232.396} C_DIS
LIN {X 0.001,Y -155.555,Z 1293.276,A 0.000,B 0.000,C 90.000,E1 229.703} C_DIS
LIN {X -0.064,Y -151.845,Z 1293.251,A 0.000,B 0.000,C 90.000,E1 225.243} C_DIS
LIN {X -0.050,Y -150.064,Z 1293.236,A 0.000,B 0.000,C 90.000,E1 222.528} C_DIS
LIN {X -0.016,Y -146.873,Z 1293.211,A 0.000,B 0.000,C 90.000,E1 217.971} C_DIS
LIN {X -0.027,Y -145.458,Z 1293.196,A 0.000,B 0.000,C 90.000,E1 215.231} C_DIS
LIN {X 0.087,Y -142.874,Z 1293.170,A 0.000,B 0.000,C 90.000,E1 210.590} C_DIS
LIN {X 0.013,Y -141.492,Z 1293.150,A 0.000,B 0.000,C 90.000,E1 206.924} C_DIS
LIN {X -0.002,Y -139.385,Z 1293.114,A 0.000,B 0.000,C 90.000,E1 200.429} C_DIS
LIN {X -0.014,Y -138.841,Z 1293.098,A 0.000,B 0.000,C 90.000,E1 197.638} C_DIS
LIN {X 0.046,Y -138.353,Z 1293.056,A 0.000,B 0.000,C 90.000,E1 190.141} C_DIS
LIN {X 0.042,Y -139.520,Z 1293.005,A 0.000,B 0.000,C 90.000,E1 180.802} C_DIS
LIN {X -0.017,Y -141.181,Z 1292.974,A 0.000,B 0.000,C 90.000,E1 175.241} C_DIS
LIN {X -0.047,Y -142.559,Z 1292.958,A 0.000,B 0.000,C 90.000,E1 172.470} C_DIS
LIN {X 0.019,Y -144.841,Z 1292.932,A 0.000,B 0.000,C 90.000,E1 167.825} C_DIS
LIN {X 0.006,Y -147.464,Z 1292.912,A 0.000,B 0.000,C 90.000,E1 164.157} C_DIS
LIN {X 0.033,Y -150.048,Z 1292.892,A 0.000,B 0.000,C 90.000,E1 160.496} C_DIS
LIN {X 0.038,Y -153.390,Z 1292.872,A 0.000,B 0.000,C 90.000,E1 156.869} C_DIS
LIN {X -0.055,Y -155.922,Z 1292.857,A 0.000,B 0.000,C 90.000,E1 154.204} C_DIS
LIN {X 0.059,Y -159.787,Z 1292.837,A 0.000,B 0.000,C 90.000,E1 150.589} C_DIS
LIN {X -0.094,Y -162.027,Z 1292.827,A 0.000,B 0.000,C 90.000,E1 148.869} C_DIS
LIN {X 0.019,Y -166.222,Z 1292.807,A 0.000,B 0.000,C 90.000,E1 145.308} C_DIS
LIN {X 0.021,Y -171.238,Z 1292.788,A 0.000,B 0.000,C 90.000,E1 141.823} C_DIS
LIN {X -0.056,Y -176.126,Z 1292.769,A 0.000,B 0.000,C 90.000,E1 138.405} C_DIS
LIN {X 0.061,Y -180.392,Z 1292.755,A 0.000,B 0.000,C 90.000,E1 135.810} C_DIS
LIN {X 0.037,Y -185.799,Z 1292.736,A 0.000,B 0.000,C 90.000,E1 132.447} C_DIS
LIN {X 0.092,Y -190.416,Z 1292.722,A 0.000,B 0.000,C 90.000,E1 129.930} C_DIS
LIN {X -0.016,Y -197.741,Z 1292.699,A 0.000,B 0.000,C 90.000,E1 125.851} C_DIS
LIN {X -0.009,Y -199.653,Z 1292.694,A 0.000,B 0.000,C 90.000,E1 124.898} C_DIS
LIN {X -0.050,Y -309.145,Z 1292.694,A 0.000,B 0.000,C 90.000,E1 124.898} C_DIS
LIN {X 0.112,Y -311.774,Z 1292.694,A 0.000,B 0.000,C 90.000,E1 124.818} C_DIS
LIN {X -0.014,Y -317.135,Z 1292.692,A 0.000,B 0.000,C 90.000,E1 124.532} C_DIS
LIN {X 0.120,Y -320.056,Z 1292.690,A 0.000,B 0.000,C 90.000,E1 124.199} C_DIS
LIN {X 0.087,Y -322.061,Z 1292.688,A 0.000,B 0.000,C 90.000,E1 123.913} C_DIS
LIN {X 0.053,Y -323.628,Z 1292.687,A 0.000,B 0.000,C 90.000,E1 123.627} C_DIS
LIN {X -0.042,Y -326.087,Z 1292.683,A 0.000,B 0.000,C 90.000,E1 123.007} C_DIS
LIN {X -0.048,Y -336.641,Z 1292.668,A 0.000,B 0.000,C 90.000,E1 120.178} C_DIS
LIN {X 0.041,Y -348.548,Z 1292.652,A 0.000,B 0.000,C 90.000,E1 117.385} C_DIS
LIN {X 0.173,Y -361.909,Z 1292.637,A 0.000,B 0.000,C 90.000,E1 114.643} C_DIS
LIN {X 0.142,Y -375.102,Z 1292.624,A 0.000,B 0.000,C 90.000,E1 112.280} C_DIS
LIN {X -0.059,Y -389.630,Z 1292.611,A 0.000,B 0.000,C 90.000,E1 109.993} C_DIS
LIN {X 0.193,Y -405.592,Z 1292.598,A 0.000,B 0.000,C 90.000,E1 107.692} C_DIS
LIN {X 0.218,Y -423.102,Z 1292.586,A 0.000,B 0.000,C 90.000,E1 105.481} C_DIS
LIN {X 0.061,Y -442.253,Z 1292.574,A 0.000,B 0.000,C 90.000,E1 103.355} C_DIS
LIN {X -0.079,Y -462.350,Z 1292.563,A 0.000,B 0.000,C 90.000,E1 101.366} C_DIS
LIN {X -0.018,Y -477.626,Z 1292.555,A 0.000,B 0.000,C 90.000,E1 99.962} C_DIS
LIN {X 0.065,Y -479.482,Z 1292.554,A 0.000,B 0.000,C 90.000,E1 99.726} C_DIS
LIN {X -0.141,Y -481.046,Z 1292.553,A 0.000,B 0.000,C 90.000,E1 99.500} C_DIS
LIN {X 0.208,Y -482.216,Z 1292.551,A 0.000,B 0.000,C 90.000,E1 99.208} C_DIS
LIN {X -0.103,Y -483.625,Z 1292.548,A 0.000,B 0.000,C 90.000,E1 98.746} C_DIS
LIN {X 0.142,Y -483.997,Z 1292.546,A 0.000,B 0.000,C 90.000,E1 98.219} C_DIS
LIN {X -0.155,Y -483.390,Z 1292.543,A 0.000,B 0.000,C 90.000,E1 97.757} C_DIS
LIN {X 0.030,Y -481.710,Z 1292.540,A 0.000,B 0.000,C 90.000,E1 97.239} C_DIS
LIN {X -0.089,Y -480.373,Z 1292.539,A 0.000,B 0.000,C 90.000,E1 97.004} C_DIS
LIN {X 0.231,Y -472.838,Z 1292.533,A 0.000,B 0.000,C 90.000,E1 95.967} C_DIS
LIN {X -0.115,Y -453.462,Z 1292.518,A 0.000,B 0.000,C 90.000,E1 93.212} C_DIS
LIN {X -0.066,Y -438.417,Z 1292.505,A 0.000,B 0.000,C 90.000,E1 90.859} C_DIS
LIN {X -0.147,Y -421.923,Z 1292.488,A 0.000,B 0.000,C 90.000,E1 87.936} C_DIS
LIN {X -0.126,Y -410.367,Z 1292.476,A 0.000,B 0.000,C 90.000,E1 85.755} C_DIS
LIN {X 0.003,Y -400.189,Z 1292.466,A 0.000,B 0.000,C 90.000,E1 83.799} C_DIS
LIN {X -0.039,Y -389.879,Z 1292.455,A 0.000,B 0.000,C 90.000,E1 81.837} C_DIS
LIN {X 0.164,Y -380.741,Z 1292.445,A 0.000,B 0.000,C 90.000,E1 80.095} C_DIS
LIN {X -0.172,Y -371.322,Z 1292.435,A 0.000,B 0.000,C 90.000,E1 78.409} C_DIS
LIN {X -0.159,Y -361.605,Z 1292.426,A 0.000,B 0.000,C 90.000,E1 76.645} C_DIS
LIN {X 0.109,Y -351.696,Z 1292.416,A 0.000,B 0.000,C 90.000,E1 74.810} C_DIS
LIN {X -0.143,Y -340.106,Z 1292.404,A 0.000,B 0.000,C 90.000,E1 72.725} C_DIS
LIN {X -0.105,Y -328.612,Z 1292.392,A 0.000,B 0.000,C 90.000,E1 70.550} C_DIS
LIN {X 0.010,Y -312.994,Z 1292.374,A 0.000,B 0.000,C 90.000,E1 67.358} C_DIS
LIN {X 0.004,Y -298.648,Z 1292.356,A 0.000,B 0.000,C 90.000,E1 64.101} C_DIS
LIN {X 0.012,Y -289.764,Z 1292.343,A 0.000,B 0.000,C 90.000,E1 61.769} C_DIS
LIN {X -0.088,Y -279.856,Z 1292.326,A 0.000,B 0.000,C 90.000,E1 58.742} C_DIS
LIN {X 0.073,Y -270.003,Z 1292.307,A 0.000,B 0.000,C 90.000,E1 55.261} C_DIS
LIN {X 0.106,Y -260.922,Z 1292.288,A 0.000,B 0.000,C 90.000,E1 51.743} C_DIS
LIN {X -0.084,Y -253.930,Z 1292.272,A 0.000,B 0.000,C 90.000,E1 48.933} C_DIS
LIN {X -0.136,Y -247.180,Z 1292.256,A 0.000,B 0.000,C 90.000,E1 46.053} C_DIS
LIN {X -0.058,Y -239.119,Z 1292.235,A 0.000,B 0.000,C 90.000,E1 42.366} C_DIS
LIN {X -0.001,Y -231.806,Z 1292.215,A 0.000,B 0.000,C 90.000,E1 38.624} C_DIS
LIN {X 0.087,Y -225.361,Z 1292.194,A 0.000,B 0.000,C 90.000,E1 34.818} C_DIS
LIN {X 0.015,Y -219.760,Z 1292.172,A 0.000,B 0.000,C 90.000,E1 31.003} C_DIS
LIN {X 0.005,Y -214.947,Z 1292.151,A 0.000,B 0.000,C 90.000,E1 27.129} C_DIS
LIN {X 0.066,Y -209.836,Z 1292.125,A 0.000,B 0.000,C 90.000,E1 22.408} C_DIS
LIN {X -0.013,Y -206.134,Z 1292.103,A 0.000,B 0.000,C 90.000,E1 18.471} C_DIS
LIN {X 0.105,Y -202.303,Z 1292.076,A 0.000,B 0.000,C 90.000,E1 13.647} C_DIS
LIN {X -0.031,Y -198.987,Z 1292.045,A 0.000,B 0.000,C 90.000,E1 8.049} C_DIS
LIN {X 0.000,Y -196.762,Z 1292.000,A 0.000,B 0.000,C 90.000,E1 360.000} C_DIS
LIN {X 0.080,Y -198.361,Z 1291.948,A 0.000,B 0.000,C 90.000,E1 350.566} C_DIS
LIN {X -0.030,Y -201.802,Z 1291.916,A 0.000,B 0.000,C 90.000,E1 344.936} C_DIS
LIN {X -0.012,Y -205.950,Z 1291.890,A 0.000,B 0.000,C 90.000,E1 340.115} C_DIS
LIN {X 0.117,Y -210.228,Z 1291.867,A 0.000,B 0.000,C 90.000,E1 336.102} C_DIS
LIN {X -0.141,Y -215.277,Z 1291.845,A 0.000,B 0.000,C 90.000,E1 332.231} C_DIS
LIN {X 0.064,Y -221.130,Z 1291.824,A 0.000,B 0.000,C 90.000,E1 328.280} C_DIS
LIN {X -0.132,Y -227.795,Z 1291.802,A 0.000,B 0.000,C 90.000,E1 324.482} C_DIS
LIN {X 0.058,Y -235.413,Z 1291.781,A 0.000,B 0.000,C 90.000,E1 320.642} C_DIS
LIN {X 0.079,Y -244.067,Z 1291.761,A 0.000,B 0.000,C 90.000,E1 316.905} C_DIS
LIN {X 0.009,Y -253.996,Z 1291.740,A 0.000,B 0.000,C 90.000,E1 313.257} C_DIS
LIN {X -0.011,Y -261.994,Z 1291.726,A 0.000,B 0.000,C 90.000,E1 310.744} C_DIS
LIN {X -0.039,Y -269.795,Z 1291.714,A 0.000,B 0.000,C 90.000,E1 308.624} C_DIS
LIN {X 0.024,Y -280.083,Z 1291.701,A 0.000,B 0.000,C 90.000,E1 306.171} C_DIS
LIN {X 0.018,Y -290.077,Z 1291.690,A 0.000,B 0.000,C 90.000,E1 304.119} C_DIS
LIN {X -0.117,Y -303.200,Z 1291.677,A 0.000,B 0.000,C 90.000,E1 301.799} C_DIS
LIN {X 0.032,Y -313.790,Z 1291.667,A 0.000,B 0.000,C 90.000,E1 300.129} C_DIS
LIN {X -0.048,Y -330.281,Z 1291.655,A 0.000,B 0.000,C 90.000,E1 297.897} C_DIS
LIN {X 0.059,Y -353.227,Z 1291.640,A 0.000,B 0.000,C 90.000,E1 295.103} C_DIS
LIN {X -0.198,Y -366.272,Z 1291.631,A 0.000,B 0.000,C 90.000,E1 293.643} C_DIS
LIN {X 0.099,Y -378.712,Z 1291.623,A 0.000,B 0.000,C 90.000,E1 292.153} C_DIS
LIN {X -0.100,Y -391.002,Z 1291.615,A 0.000,B 0.000,C 90.000,E1 290.737} C_DIS
LIN {X 0.162,Y -408.288,Z 1291.604,A 0.000,B 0.000,C 90.000,E1 288.725} C_DIS
LIN {X 0.091,Y -418.354,Z 1291.598,A 0.000,B 0.000,C 90.000,E1 287.638} C_DIS
LIN {X 0.064,Y -428.045,Z 1291.592,A 0.000,B 0.000,C 90.000,E1 286.551} C_DIS
LIN {X 0.027,Y -436.974,Z 1291.586,A 0.000,B 0.000,C 90.000,E1 285.481} C_DIS
LIN {X -0.227,Y -442.821,Z 1291.582,A 0.000,B 0.000,C 90.000,E1 284.717} C_DIS
LIN {X 0.109,Y -447.920,Z 1291.577,A 0.000,B 0.000,C 90.000,E1 283.883} C_DIS
LIN {X -0.045,Y -452.391,Z 1291.573,A 0.000,B 0.000,C 90.000,E1 283.119} C_DIS
LIN {X -0.168,Y -456.321,Z 1291.568,A 0.000,B 0.000,C 90.000,E1 282.355} C_DIS
LIN {X -0.080,Y -458.576,Z 1291.566,A 0.000,B 0.000,C 90.000,E1 281.827} C_DIS
LIN {X 0.022,Y -460.602,Z 1291.563,A 0.000,B 0.000,C 90.000,E1 281.299} C_DIS
LIN {X 0.044,Y -462.330,Z 1291.560,A 0.000,B 0.000,C 90.000,E1 280.782} C_DIS
LIN {X 0.166,Y -463.716,Z 1291.557,A 0.000,B 0.000,C 90.000,E1 280.254} C_DIS
LIN {X -0.163,Y -464.782,Z 1291.554,A 0.000,B 0.000,C 90.000,E1 279.782} C_DIS
LIN {X -0.106,Y -465.426,Z 1291.551,A 0.000,B 0.000,C 90.000,E1 279.265} C_DIS
LIN {X -0.038,Y -465.659,Z 1291.549,A 0.000,B 0.000,C 90.000,E1 278.746} C_DIS
LIN {X 0.104,Y -465.494,Z 1291.546,A 0.000,B 0.000,C 90.000,E1 278.219} C_DIS
LIN {X 0.178,Y -464.852,Z 1291.543,A 0.000,B 0.000,C 90.000,E1 277.701} C_DIS
LIN {X -0.208,Y -463.713,Z 1291.540,A 0.000,B 0.000,C 90.000,E1 277.239} C_DIS
LIN {X -0.136,Y -462.070,Z 1291.537,A 0.000,B 0.000,C 90.000,E1 276.720} C_DIS
LIN {X 0.209,Y -458.843,Z 1291.533,A 0.000,B 0.000,C 90.000,E1 275.910} C_DIS
LIN {X -0.202,Y -456.207,Z 1291.530,A 0.000,B 0.000,C 90.000,E1 275.448} C_DIS
LIN {X -0.214,Y -453.124,Z 1291.527,A 0.000,B 0.000,C 90.000,E1 274.935} C_DIS
LIN {X -0.202,Y -449.326,Z 1291.524,A 0.000,B 0.000,C 90.000,E1 274.416} C_DIS
LIN {X -0.210,Y -444.650,Z 1291.521,A 0.000,B 0.000,C 90.000,E1 273.898} C_DIS
LIN {X -0.015,Y -441.924,Z 1291.520,A 0.000,B 0.000,C 90.000,E1 273.612} C_DIS
LIN {X 0.186,Y -435.778,Z 1291.517,A 0.000,B 0.000,C 90.000,E1 273.094} C_DIS
LIN {X 0.015,Y -429.387,Z 1291.515,A 0.000,B 0.000,C 90.000,E1 272.694} C_DIS
LIN {X -0.168,Y -422.464,Z 1291.513,A 0.000,B 0.000,C 90.000,E1 272.350} C_DIS
LIN {X 0.143,Y -415.529,Z 1291.511,A 0.000,B 0.000,C 90.000,E1 272.007} C_DIS
LIN {X -0.020,Y -408.454,Z 1291.510,A 0.000,B 0.000,C 90.000,E1 271.776} C_DIS
LIN {X 0.123,Y -401.387,Z 1291.509,A 0.000,B 0.000,C 90.000,E1 271.547} C_DIS
LIN {X -0.003,Y -390.536,Z 1291.507,A 0.000,B 0.000,C 90.000,E1 271.318} C_DIS
LIN {X -0.093,Y -377.889,Z 1291.506,A 0.000,B 0.000,C 90.000,E1 271.146} C_DIS
LIN {X 0.044,Y -365.281,Z 1291.506,A 0.000,B 0.000,C 90.000,E1 271.031} C_DIS
LIN {X -0.104,Y -357.040,Z 1291.506,A 0.000,B 0.000,C 90.000,E1 271.031} C_DIS
LIN {X -0.078,Y -181.454,Z 1291.506,A 0.000,B 0.000,C 90.000,E1 271.031} C_DIS
LIN {X 0.060,Y -181.576,Z 1291.501,A 0.000,B 0.000,C 90.000,E1 270.115} C_DIS
LIN {X 0.047,Y -180.878,Z 1291.473,A 0.000,B 0.000,C 90.000,E1 265.065} C_DIS
LIN {X -0.073,Y -178.996,Z 1291.445,A 0.000,B 0.000,C 90.000,E1 260.038} C_DIS
LIN {X 0.022,Y -178.584,Z 1291.440,A 0.000,B 0.000,C 90.000,E1 259.162} C_DIS
LIN {X -0.085,Y -175.636,Z 1291.411,A 0.000,B 0.000,C 90.000,E1 254.102} C_DIS
LIN {X -0.019,Y -172.356,Z 1291.388,A 0.000,B 0.000,C 90.000,E1 249.806} C_DIS
LIN {X -0.064,Y -171.141,Z 1291.378,A 0.000,B 0.000,C 90.000,E1 248.103} C_DIS
LIN {X -0.019,Y -167.445,Z 1291.354,A 0.000,B 0.000,C 90.000,E1 243.768} C_DIS
LIN {X 0.063,Y -166.841,Z 1291.349,A 0.000,B 0.000,C 90.000,E1 242.871} C_DIS
LIN {X -0.020,Y -162.825,Z 1291.325,A 0.000,B 0.000,C 90.000,E1 238.535} C_DIS
LIN {X 0.044,Y -161.510,Z 1291.315,A 0.000,B 0.000,C 90.000,E1 236.755} C_DIS
LIN {X -0.003,Y -157.508,Z 1291.291,A 0.000,B 0.000,C 90.000,E1 232.351} C_DIS
LIN {X 0.031,Y -155.530,Z 1291.276,A 0.000,B 0.000,C 90.000,E1 229.666} C_DIS
LIN {X 0.080,Y -151.827,Z 1291.251,A 0.000,B 0.000,C 90.000,E1 225.162} C_DIS
LIN {X -0.009,Y -150.042,Z 1291.236,A 0.000,B 0.000,C 90.000,E1 222.486} C_DIS
LIN {X 0.005,Y -146.857,Z 1291.211,A 0.000,B 0.000,C 90.000,E1 217.935} C_DIS
LIN {X 0.024,Y -145.442,Z 1291.196,A 0.000,B 0.000,C 90.000,E1 215.185} C_DIS
LIN {X 0.018,Y -142.862,Z 1291.170,A 0.000,B 0.000,C 90.000,E1 210.590} C_DIS
LIN {X 0.071,Y -141.479,Z 1291.149,A 0.000,B 0.000,C 90.000,E1 206.873} C_DIS
LIN {X -0.070,Y -139.381,Z 1291.113,A 0.000,B 0.000,C 90.000,E1 200.429} C_DIS
LIN {X 0.051,Y -138.834,Z 1291.098,A 0.000,B 0.000,C 90.000,E1 197.583} C_DIS
LIN {X -0.021,Y -138.354,Z 1291.056,A 0.000,B 0.000,C 90.000,E1 190.141} C_DIS
LIN {X -0.025,Y -139.524,Z 1291.004,A 0.000,B 0.000,C 90.000,E1 180.802} C_DIS
LIN {X 0.055,Y -141.193,Z 1290.973,A 0.000,B 0.000,C 90.000,E1 175.184} C_DIS
LIN {X 0.027,Y -142.570,Z 1290.958,A 0.000,B 0.000,C 90.000,E1 172.413} C_DIS
LIN {X -0.018,Y -144.857,Z 1290.932,A 0.000,B 0.000,C 90.000,E1 167.813} C_DIS
LIN {X -0.063,Y -147.483,Z 1290.912,A 0.000,B 0.000,C 90.000,E1 164.157} C_DIS
LIN {X -0.037,Y -150.069,Z 1290.892,A 0.000,B 0.000,C 90.000,E1 160.496} C_DIS
LIN {X -0.033,Y -153.418,Z 1290.871,A 0.000,B 0.000,C 90.000,E1 156.869} C_DIS
LIN {X 0.015,Y -156.839,Z 1290.851,A 0.000,B 0.000,C 90.000,E1 153.256} C_DIS
LIN {X 0.087,Y -160.918,Z 1290.832,A 0.000,B 0.000,C 90.000,E1 149.665} C_DIS
LIN {X 0.031,Y -163.043,Z 1290.822,A 0.000,B 0.000,C 90.000,E1 147.916} C_DIS
LIN {X 0.036,Y -167.435,Z 1290.802,A 0.000,B 0.000,C 90.000,E1 144.402} C_DIS
LIN {X -0.055,Y -171.273,Z 1290.788,A 0.000,B 0.000,C 90.000,E1 141.823} C_DIS
LIN {X -0.016,Y -176.165,Z 1290.769,A 0.000,B 0.000,C 90.000,E1 138.366} C_DIS
LIN {X -0.018,Y -180.437,Z 1290.755,A 0.000,B 0.000,C 90.000,E1 135.810} C_DIS
LIN {X -0.043,Y -185.842,Z 1290.736,A 0.000,B 0.000,C 90.000,E1 132.447} C_DIS
LIN {X 0.010,Y -190.464,Z 1290.722,A 0.000,B 0.000,C 90.000,E1 129.930} C_DIS
LIN {X -0.085,Y -196.217,Z 1290.703,A 0.000,B 0.000,C 90.000,E1 126.664} C_DIS
LIN {X -0.070,Y -199.689,Z 1290.694,A 0.000,B 0.000,C 90.000,E1 124.898} C_DIS
LIN {X -0.144,Y -309.060,Z 1290.694,A 0.000,B 0.000,C 90.000,E1 124.898} C_DIS
LIN {X -0.018,Y -311.993,Z 1290.693,A 0.000,B 0.000,C 90.000,E1 124.818} C_DIS
LIN {X 0.115,Y -317.241,Z 1290.692,A 0.000,B 0.000,C 90.000,E1 124.485} C_DIS
LIN {X -0.014,Y -320.142,Z 1290.690,A 0.000,B 0.000,C 90.000,E1 124.199} C_DIS
LIN {X -0.055,Y -322.146,Z 1290.688,A 0.000,B 0.000,C 90.000,E1 123.913} C_DIS
LIN {X -0.098,Y -323.711,Z 1290.687,A 0.000,B 0.000,C 90.000,E1 123.627} C_DIS
LIN {X 0.079,Y -326.160,Z 1290.683,A 0.000,B 0.000,C 90.000,E1 122.959} C_DIS
LIN {X 0.087,Y -336.725,Z 1290.667,A 0.000,B 0.000,C 90.000,E1 120.129} C_DIS
LIN {X -0.118,Y -348.646,Z 1290.652,A 0.000,B 0.000,C 90.000,E1 117.385} C_DIS
LIN {X 0.011,Y -362.021,Z 1290.637,A 0.000,B 0.000,C 90.000,E1 114.643} C_DIS
LIN {X -0.023,Y -375.227,Z 1290.624,A 0.000,B 0.000,C 90.000,E1 112.280} C_DIS
LIN {X 0.138,Y -389.768,Z 1290.611,A 0.000,B 0.000,C 90.000,E1 109.939} C_DIS
LIN {X 0.021,Y -405.747,Z 1290.598,A 0.000,B 0.000,C 90.000,E1 107.692} C_DIS
LIN {X 0.042,Y -423.274,Z 1290.586,A 0.000,B 0.000,C 90.000,E1 105.481} C_DIS
LIN {X -0.117,Y -442.442,Z 1290.574,A 0.000,B 0.000,C 90.000,E1 103.355} C_DIS
LIN {X -0.250,Y -462.545,Z 1290.563,A 0.000,B 0.000,C 90.000,E1 101.366} C_DIS
LIN {X 0.198,Y -475.401,Z 1290.557,A 0.000,B 0.000,C 90.000,E1 100.141} C_DIS
LIN {X -0.185,Y -477.761,Z 1290.555,A 0.000,B 0.000,C 90.000,E1 99.962} C_DIS
LIN {X -0.101,Y -479.551,Z 1290.554,A 0.000,B 0.000,C 90.000,E1 99.726} C_DIS
LIN {X 0.168,Y -481.063,Z 1290.553,A 0.000,B 0.000,C 90.000,E1 99.443} C_DIS
LIN {X 0.042,Y -482.192,Z 1290.551,A 0.000,B 0.000,C 90.000,E1 99.208} C_DIS
LIN {X -0.269,Y -483.537,Z 1290.548,A 0.000,B 0.000,C 90.000,E1 98.746} C_DIS
LIN {X -0.025,Y -483.850,Z 1290.546,A 0.000,B 0.000,C 90.000,E1 98.219} C_DIS
LIN {X 0.157,Y -483.187,Z 1290.543,A 0.000,B 0.000,C 90.000,E1 97.701} C_DIS
LIN {X -0.137,Y -481.439,Z 1290.540,A 0.000,B 0.000,C 90.000,E1 97.239} C_DIS
LIN {X 0.221,Y -480.057,Z 1290.539,A 0.000,B 0.000,C 90.000,E1 96.947} C_DIS
LIN {X -0.215,Y -465.265,Z 1290.528,A 0.000,B 0.000,C 90.000,E1 94.992} C_DIS
LIN {X 0.167,Y -453.120,Z 1290.518,A 0.000,B 0.000,C 90.000,E1 93.154} C_DIS
LIN {X 0.197,Y -438.085,Z 1290.505,A 0.000,B 0.000,C 90.000,E1 90.802} C_DIS
LIN {X -0.027,Y -423.035,Z 1290.490,A 0.000,B 0.000,C 90.000,E1 88.165} C_DIS
LIN {X -0.010,Y -411.455,Z 1290.478,A 0.000,B 0.000,C 90.000,E1 85.988} C_DIS
LIN {X 0.135,Y -401.316,Z 1290.467,A 0.000,B 0.000,C 90.000,E1 84.033} C_DIS
LIN {X 0.156,Y -391.033,Z 1290.456,A 0.000,B 0.000,C 90.000,E1 82.064} C_DIS
LIN {X -0.058,Y -381.959,Z 1290.447,A 0.000,B 0.000,C 90.000,E1 80.387} C_DIS
LIN {X 0.071,Y -372.589,Z 1290.437,A 0.000,B 0.000,C 90.000,E1 78.634} C_DIS
LIN {X 0.026,Y -362.914,Z 1290.427,A 0.000,B 0.000,C 90.000,E1 76.881} C_DIS
LIN {X -0.027,Y -353.046,Z 1290.417,A 0.000,B 0.000,C 90.000,E1 75.102} C_DIS
LIN {X 0.089,Y -341.449,Z 1290.405,A 0.000,B 0.000,C 90.000,E1 72.960} C_DIS
LIN {X 0.015,Y -328.315,Z 1290.392,A 0.000,B 0.000,C 90.000,E1 70.496} C_DIS
LIN {X -0.179,Y -312.737,Z 1290.374,A 0.000,B 0.000,C 90.000,E1 67.358} C_DIS
LIN {X -0.071,Y -299.800,Z 1290.358,A 0.000,B 0.000,C 90.000,E1 64.409} C_DIS
LIN {X -0.166,Y -290.776,Z 1290.345,A 0.000,B 0.000,C 90.000,E1 62.103} C_DIS
LIN {X 0.176,Y -281.756,Z 1290.330,A 0.000,B 0.000,C 90.000,E1 59.331} C_DIS
LIN {X 0.019,Y -271.742,Z 1290.311,A 0.000,B 0.000,C 90.000,E1 55.928} C_DIS
LIN {X 0.008,Y -262.481,Z 1290.291,A 0.000,B 0.000,C 90.000,E1 52.431} C_DIS
LIN {X 0.018,Y -255.441,Z 1290.276,A 0.000,B 0.000,C 90.000,E1 49.585} C_DIS
LIN {X 0.020,Y -248.637,Z 1290.260,A 0.000,B 0.000,C 90.000,E1 46.701} C_DIS
LIN {X -0.037,Y -240.461,Z 1290.239,A 0.000,B 0.000,C 90.000,E1 43.056} C_DIS
LIN {X 0.027,Y -232.982,Z 1290.219,A 0.000,B 0.000,C 90.000,E1 39.322} C_DIS
LIN {X 0.142,Y -226.372,Z 1290.198,A 0.000,B 0.000,C 90.000,E1 35.518} C_DIS
LIN {X 0.031,Y -220.565,Z 1290.176,A 0.000,B 0.000,C 90.000,E1 31.720} C_DIS
LIN {X 0.040,Y -215.573,Z 1290.155,A 0.000,B 0.000,C 90.000,E1 27.847} C_DIS
LIN {X 0.021,Y -210.285,Z 1290.129,A 0.000,B 0.000,C 90.000,E1 23.153} C_DIS
LIN {X 0.019,Y -207.202,Z 1290.111,A 0.000,B 0.000,C 90.000,E1 19.993} C_DIS
LIN {X 0.100,Y -203.112,Z 1290.085,A 0.000,B 0.000,C 90.000,E1 15.190} C_DIS
LIN {X -0.081,Y -199.437,Z 1290.053,A 0.000,B 0.000,C 90.000,E1 9.613} C_DIS
LIN {X 0.012,Y -196.813,Z 1290.013,A 0.000,B 0.000,C 90.000,E1 2.293} C_DIS
LIN {X 0.065,Y -198.220,Z 1289.948,A 0.000,B 0.000,C 90.000,E1 350.566} C_DIS
LIN {X -0.051,Y -201.747,Z 1289.916,A 0.000,B 0.000,C 90.000,E1 344.936} C_DIS
LIN {X -0.034,Y -205.919,Z 1289.890,A 0.000,B 0.000,C 90.000,E1 340.115} C_DIS
LIN {X 0.093,Y -210.231,Z 1289.867,A 0.000,B 0.000,C 90.000,E1 336.102} C_DIS
LIN {X 0.125,Y -215.303,Z 1289.845,A 0.000,B 0.000,C 90.000,E1 332.153} C_DIS
LIN {X 0.040,Y -221.156,Z 1289.824,A 0.000,B 0.000,C 90.000,E1 328.280} C_DIS
LIN {X 0.028,Y -227.824,Z 1289.802,A 0.000,B 0.000,C 90.000,E1 324.436} C_DIS
LIN {X 0.034,Y -235.454,Z 1289.781,A 0.000,B 0.000,C 90.000,E1 320.642} C_DIS
LIN {X 0.055,Y -244.081,Z 1289.761,A 0.000,B 0.000,C 90.000,E1 316.905} C_DIS
LIN {X -0.023,Y -252.951,Z 1289.742,A 0.000,B 0.000,C 90.000,E1 313.623} C_DIS
LIN {X 0.081,Y -259.595,Z 1289.730,A 0.000,B 0.000,C 90.000,E1 311.434} C_DIS
LIN {X 0.033,Y -268.421,Z 1289.716,A 0.000,B 0.000,C 90.000,E1 308.955} C_DIS
LIN {X 0.062,Y -278.532,Z 1289.703,A 0.000,B 0.000,C 90.000,E1 306.503} C_DIS
LIN {X -0.106,Y -286.615,Z 1289.693,A 0.000,B 0.000,C 90.000,E1 304.818} C_DIS
LIN {X 0.098,Y -295.496,Z 1289.684,A 0.000,B 0.000,C 90.000,E1 303.086} C_DIS
LIN {X -0.134,Y -305.206,Z 1289.675,A 0.000,B 0.000,C 90.000,E1 301.465} C_DIS
LIN {X 0.054,Y -316.008,Z 1289.666,A 0.000,B 0.000,C 90.000,E1 299.795} C_DIS
LIN {X -0.139,Y -332.752,Z 1289.653,A 0.000,B 0.000,C 90.000,E1 297.590} C_DIS
LIN {X 0.058,Y -353.333,Z 1289.639,A 0.000,B 0.000,C 90.000,E1 295.079} C_DIS
LIN {X -0.017,Y -366.399,Z 1289.631,A 0.000,B 0.000,C 90.000,E1 293.590} C_DIS
LIN {X 0.110,Y -379.074,Z 1289.623,A 0.000,B 0.000,C 90.000,E1 292.099} C_DIS
LIN {X 0.083,Y -391.326,Z 1289.615,A 0.000,B 0.000,C 90.000,E1 290.663} C_DIS
LIN {X 0.068,Y -416.242,Z 1289.599,A 0.000,B 0.000,C 90.000,E1 287.873} C_DIS
LIN {X -0.087,Y -425.975,Z 1289.593,A 0.000,B 0.000,C 90.000,E1 286.804} C_DIS
LIN {X 0.102,Y -432.952,Z 1289.589,A 0.000,B 0.000,C 90.000,E1 285.969} C_DIS
LIN {X -0.066,Y -439.280,Z 1289.584,A 0.000,B 0.000,C 90.000,E1 285.190} C_DIS
LIN {X 0.239,Y -444.910,Z 1289.580,A 0.000,B 0.000,C 90.000,E1 284.356} C_DIS
LIN {X 0.058,Y -449.802,Z 1289.576,A 0.000,B 0.000,C 90.000,E1 283.592} C_DIS
LIN {X -0.085,Y -454.074,Z 1289.571,A 0.000,B 0.000,C 90.000,E1 282.827} C_DIS
LIN {X -0.187,Y -457.793,Z 1289.567,A 0.000,B 0.000,C 90.000,E1 282.063} C_DIS
LIN {X 0.188,Y -460.871,Z 1289.563,A 0.000,B 0.000,C 90.000,E1 281.243} C_DIS
LIN {X -0.243,Y -462.570,Z 1289.560,A 0.000,B 0.000,C 90.000,E1 280.782} C_DIS
LIN {X -0.119,Y -463.927,Z 1289.557,A 0.000,B 0.000,C 90.000,E1 280.254} C_DIS
LIN {X 0.010,Y -464.956,Z 1289.554,A 0.000,B 0.000,C 90.000,E1 279.726} C_DIS
LIN {X 0.070,Y -465.614,Z 1289.551,A 0.000,B 0.000,C 90.000,E1 279.208} C_DIS
LIN {X 0.140,Y -465.851,Z 1289.548,A 0.000,B 0.000,C 90.000,E1 278.690} C_DIS
LIN {X -0.178,Y -465.684,Z 1289.546,A 0.000,B 0.000,C 90.000,E1 278.219} C_DIS
LIN {X -0.103,Y -464.995,Z 1289.543,A 0.000,B 0.000,C 90.000,E1 277.701} C_DIS
LIN {X -0.027,Y -463.823,Z 1289.540,A 0.000,B 0.000,C 90.000,E1 277.182} C_DIS
LIN {X 0.047,Y -462.194,Z 1289.537,A 0.000,B 0.000,C 90.000,E1 276.663} C_DIS
LIN {X -0.064,Y -458.977,Z 1289.533,A 0.000,B 0.000,C 90.000,E1 275.910} C_DIS
LIN {X -0.019,Y -456.368,Z 1289.530,A 0.000,B 0.000,C 90.000,E1 275.391} C_DIS
LIN {X -0.031,Y -453.273,Z 1289.527,A 0.000,B 0.000,C 90.000,E1 274.878} C_DIS
LIN {X -0.019,Y -449.562,Z 1289.524,A 0.000,B 0.000,C 90.000,E1 274.359} C_DIS
LIN {X -0.029,Y -444.867,Z 1289.521,A 0.000,B 0.000,C 90.000,E1 273.841} C_DIS
LIN {X 0.167,Y -442.126,Z 1289.520,A 0.000,B 0.000,C 90.000,E1 273.555} C_DIS
LIN {X -0.005,Y -436.083,Z 1289.517,A 0.000,B 0.000,C 90.000,E1 273.094} C_DIS
LIN {X -0.162,Y -429.753,Z 1289.515,A 0.000,B 0.000,C 90.000,E1 272.694} C_DIS
LIN {X 0.110,Y -422.970,Z 1289.513,A 0.000,B 0.000,C 90.000,E1 272.293} C_DIS
LIN {X -0.039,Y -415.871,Z 1289.511,A 0.000,B 0.000,C 90.000,E1 272.007} C_DIS
LIN {X -0.183,Y -408.833,Z 1289.510,A 0.000,B 0.000,C 90.000,E1 271.776} C_DIS
LIN {X 0.152,Y -398.403,Z 1289.508,A 0.000,B 0.000,C 90.000,E1 271.432} C_DIS
LIN {X -0.160,Y -391.054,Z 1289.507,A 0.000,B 0.000,C 90.000,E1 271.318} C_DIS
LIN {X 0.127,Y -378.369,Z 1289.506,A 0.000,B 0.000,C 90.000,E1 271.088} C_DIS
LIN {X -0.114,Y -365.868,Z 1289.506,A 0.000,B 0.000,C 90.000,E1 271.031} C_DIS
LIN {X 0.094,Y -356.855,Z 1289.505,A 0.000,B 0.000,C 90.000,E1 270.974} C_DIS
LIN {X 0.023,Y -181.461,Z 1289.505,A 0.000,B 0.000,C 90.000,E1 270.974} C_DIS
LIN {X -0.025,Y -181.574,Z 1289.501,A 0.000,B 0.000,C 90.000,E1 270.115} C_DIS
LIN {X -0.038,Y -180.873,Z 1289.473,A 0.000,B 0.000,C 90.000,E1 265.065} C_DIS
LIN {X 0.020,Y -178.990,Z 1289.444,A 0.000,B 0.000,C 90.000,E1 259.982} C_DIS
LIN {X 0.031,Y -177.974,Z 1289.435,A 0.000,B 0.000,C 90.000,E1 258.285} C_DIS
LIN {X 0.049,Y -175.617,Z 1289.411,A 0.000,B 0.000,C 90.000,E1 254.031} C_DIS
LIN {X 0.061,Y -172.339,Z 1289.388,A 0.000,B 0.000,C 90.000,E1 249.752} C_DIS
LIN {X 0.039,Y -171.816,Z 1289.383,A 0.000,B 0.000,C 90.000,E1 248.901} C_DIS
LIN {X 0.047,Y -170.281,Z 1289.373,A 0.000,B 0.000,C 90.000,E1 247.177} C_DIS
LIN {X -0.017,Y -166.821,Z 1289.349,A 0.000,B 0.000,C 90.000,E1 242.871} C_DIS
LIN {X -0.099,Y -162.803,Z 1289.325,A 0.000,B 0.000,C 90.000,E1 238.535} C_DIS
LIN {X -0.035,Y -161.489,Z 1289.315,A 0.000,B 0.000,C 90.000,E1 236.755} C_DIS
LIN {X 0.015,Y -157.486,Z 1289.291,A 0.000,B 0.000,C 90.000,E1 232.316} C_DIS
LIN {X -0.047,Y -155.504,Z 1289.276,A 0.000,B 0.000,C 90.000,E1 229.666} C_DIS
LIN {X 0.004,Y -151.807,Z 1289.251,A 0.000,B 0.000,C 90.000,E1 225.162} C_DIS
LIN {X 0.017,Y -150.018,Z 1289.236,A 0.000,B 0.000,C 90.000,E1 222.447} C_DIS
LIN {X 0.047,Y -146.841,Z 1289.211,A 0.000,B 0.000,C 90.000,E1 217.890} C_DIS
LIN {X -0.050,Y -145.424,Z 1289.195,A 0.000,B 0.000,C 90.000,E1 215.185} C_DIS
LIN {X -0.054,Y -142.849,Z 1289.170,A 0.000,B 0.000,C 90.000,E1 210.590} C_DIS
LIN {X -0.002,Y -141.464,Z 1289.149,A 0.000,B 0.000,C 90.000,E1 206.873} C_DIS
LIN {X -0.011,Y -139.376,Z 1289.113,A 0.000,B 0.000,C 90.000,E1 200.375} C_DIS
LIN {X -0.020,Y -138.827,Z 1289.098,A 0.000,B 0.000,C 90.000,E1 197.583} C_DIS
LIN {X 0.044,Y -138.353,Z 1289.056,A 0.000,B 0.000,C 90.000,E1 190.084} C_DIS
LIN {X 0.042,Y -139.529,Z 1289.004,A 0.000,B 0.000,C 90.000,E1 180.745} C_DIS
LIN {X -0.005,Y -141.206,Z 1288.973,A 0.000,B 0.000,C 90.000,E1 175.179} C_DIS
LIN {X -0.046,Y -142.581,Z 1288.958,A 0.000,B 0.000,C 90.000,E1 172.413} C_DIS
LIN {X 0.050,Y -144.875,Z 1288.932,A 0.000,B 0.000,C 90.000,E1 167.757} C_DIS
LIN {X 0.003,Y -147.502,Z 1288.912,A 0.000,B 0.000,C 90.000,E1 164.102} C_DIS
LIN {X 0.078,Y -150.093,Z 1288.891,A 0.000,B 0.000,C 90.000,E1 160.423} C_DIS
LIN {X -0.050,Y -153.448,Z 1288.871,A 0.000,B 0.000,C 90.000,E1 156.847} C_DIS
LIN {X -0.057,Y -157.811,Z 1288.846,A 0.000,B 0.000,C 90.000,E1 152.359} C_DIS
LIN {X -0.024,Y -162.093,Z 1288.827,A 0.000,B 0.000,C 90.000,E1 148.791} C_DIS
LIN {X 0.000,Y -166.293,Z 1288.807,A 0.000,B 0.000,C 90.000,E1 145.261} C_DIS
LIN {X -0.003,Y -171.309,Z 1288.788,A 0.000,B 0.000,C 90.000,E1 141.778} C_DIS
LIN {X 0.032,Y -176.207,Z 1288.769,A 0.000,B 0.000,C 90.000,E1 138.324} C_DIS
LIN {X -0.103,Y -180.484,Z 1288.754,A 0.000,B 0.000,C 90.000,E1 135.810} C_DIS
LIN {X 0.008,Y -185.888,Z 1288.736,A 0.000,B 0.000,C 90.000,E1 132.405} C_DIS
LIN {X -0.077,Y -190.515,Z 1288.722,A 0.000,B 0.000,C 90.000,E1 129.930} C_DIS
LIN {X 0.101,Y -196.266,Z 1288.703,A 0.000,B 0.000,C 90.000,E1 126.583} C_DIS
LIN {X -0.013,Y -199.722,Z 1288.694,A 0.000,B 0.000,C 90.000,E1 124.865} C_DIS
LIN {X 0.183,Y -309.408,Z 1288.694,A 0.000,B 0.000,C 90.000,E1 124.818} C_DIS
LIN {X -0.053,Y -314.607,Z 1288.693,A 0.000,B 0.000,C 90.000,E1 124.692} C_DIS
LIN {X -0.115,Y -317.017,Z 1288.692,A 0.000,B 0.000,C 90.000,E1 124.532} C_DIS
LIN {X -0.157,Y -320.249,Z 1288.690,A 0.000,B 0.000,C 90.000,E1 124.199} C_DIS
LIN {X 0.081,Y -322.222,Z 1288.688,A 0.000,B 0.000,C 90.000,E1 123.865} C_DIS
LIN {X 0.054,Y -323.767,Z 1288.687,A 0.000,B 0.000,C 90.000,E1 123.579} C_DIS
LIN {X -0.040,Y -326.211,Z 1288.683,A 0.000,B 0.000,C 90.000,E1 122.959} C_DIS
LIN {X -0.032,Y -336.785,Z 1288.667,A 0.000,B 0.000,C 90.000,E1 120.129} C_DIS
LIN {X 0.069,Y -348.716,Z 1288.652,A 0.000,B 0.000,C 90.000,E1 117.334} C_DIS
LIN {X -0.114,Y -362.102,Z 1288.637,A 0.000,B 0.000,C 90.000,E1 114.643} C_DIS
LIN {X -0.151,Y -375.318,Z 1288.624,A 0.000,B 0.000,C 90.000,E1 112.280} C_DIS
LIN {X 0.008,Y -389.871,Z 1288.611,A 0.000,B 0.000,C 90.000,E1 109.939} C_DIS
LIN {X -0.112,Y -405.861,Z 1288.598,A 0.000,B 0.000,C 90.000,E1 107.692} C_DIS
LIN {X -0.093,Y -423.402,Z 1288.586,A 0.000,B 0.000,C 90.000,E1 105.481} C_DIS
LIN {X 0.176,Y -442.583,Z 1288.574,A 0.000,B 0.000,C 90.000,E1 103.300} C_DIS
LIN {X 0.162,Y -462.691,Z 1288.563,A 0.000,B 0.000,C 90.000,E1 101.299} C_DIS
LIN {X 0.068,Y -475.549,Z 1288.556,A 0.000,B 0.000,C 90.000,E1 100.141} C_DIS
LIN {X 0.156,Y -477.846,Z 1288.555,A 0.000,B 0.000,C 90.000,E1 99.905} C_DIS
LIN {X 0.244,Y -479.582,Z 1288.554,A 0.000,B 0.000,C 90.000,E1 99.670} C_DIS
LIN {X 0.039,Y -481.053,Z 1288.552,A 0.000,B 0.000,C 90.000,E1 99.443} C_DIS
LIN {X -0.087,Y -482.148,Z 1288.551,A 0.000,B 0.000,C 90.000,E1 99.208} C_DIS
LIN {X 0.080,Y -483.438,Z 1288.548,A 0.000,B 0.000,C 90.000,E1 98.690} C_DIS
LIN {X -0.154,Y -483.705,Z 1288.546,A 0.000,B 0.000,C 90.000,E1 98.219} C_DIS
LIN {X 0.027,Y -482.992,Z 1288.543,A 0.000,B 0.000,C 90.000,E1 97.701} C_DIS
LIN {X 0.210,Y -481.186,Z 1288.540,A 0.000,B 0.000,C 90.000,E1 97.182} C_DIS
LIN {X 0.090,Y -479.766,Z 1288.539,A 0.000,B 0.000,C 90.000,E1 96.947} C_DIS
LIN {X 0.116,Y -464.978,Z 1288.527,A 0.000,B 0.000,C 90.000,E1 94.935} C_DIS
LIN {X -0.180,Y -451.072,Z 1288.516,A 0.000,B 0.000,C 90.000,E1 92.922} C_DIS
LIN {X 0.059,Y -437.781,Z 1288.505,A 0.000,B 0.000,C 90.000,E1 90.802} C_DIS
LIN {X 0.068,Y -419.819,Z 1288.487,A 0.000,B 0.000,C 90.000,E1 87.593} C_DIS
LIN {X 0.027,Y -408.231,Z 1288.474,A 0.000,B 0.000,C 90.000,E1 85.412} C_DIS
LIN {X 0.068,Y -399.545,Z 1288.465,A 0.000,B 0.000,C 90.000,E1 83.742} C_DIS
LIN {X 0.009,Y -389.239,Z 1288.454,A 0.000,B 0.000,C 90.000,E1 81.781} C_DIS
LIN {X -0.176,Y -380.141,Z 1288.445,A 0.000,B 0.000,C 90.000,E1 80.095} C_DIS
LIN {X -0.077,Y -370.704,Z 1288.435,A 0.000,B 0.000,C 90.000,E1 78.342} C_DIS
LIN {X -0.153,Y -360.986,Z 1288.425,A 0.000,B 0.000,C 90.000,E1 76.589} C_DIS
LIN {X 0.102,Y -351.091,Z 1288.415,A 0.000,B 0.000,C 90.000,E1 74.755} C_DIS
LIN {X -0.065,Y -339.502,Z 1288.404,A 0.000,B 0.000,C 90.000,E1 72.653} C_DIS
LIN {X -0.176,Y -326.433,Z 1288.390,A 0.000,B 0.000,C 90.000,E1 70.188} C_DIS
LIN {X -0.006,Y -311.015,Z 1288.372,A 0.000,B 0.000,C 90.000,E1 66.975} C_DIS
LIN {X 0.040,Y -299.610,Z 1288.358,A 0.000,B 0.000,C 90.000,E1 64.357} C_DIS
LIN {X 0.070,Y -290.623,Z 1288.345,A 0.000,B 0.000,C 90.000,E1 62.025} C_DIS
LIN {X 0.020,Y -281.603,Z 1288.330,A 0.000,B 0.000,C 90.000,E1 59.331} C_DIS
LIN {X 0.089,Y -271.561,Z 1288.311,A 0.000,B 0.000,C 90.000,E1 55.881} C_DIS
LIN {X 0.013,Y -262.283,Z 1288.291,A 0.000,B 0.000,C 90.000,E1 52.396} C_DIS
LIN {X 0.056,Y -255.234,Z 1288.275,A 0.000,B 0.000,C 90.000,E1 49.542} C_DIS
LIN {X 0.033,Y -248.424,Z 1288.259,A 0.000,B 0.000,C 90.000,E1 46.662} C_DIS
LIN {X -0.020,Y -240.246,Z 1288.239,A 0.000,B 0.000,C 90.000,E1 43.014} C_DIS
LIN {X 0.046,Y -232.771,Z 1288.218,A 0.000,B 0.000,C 90.000,E1 39.277} C_DIS
LIN {X -0.020,Y -226.146,Z 1288.197,A 0.000,B 0.000,C 90.000,E1 35.518} C_DIS
LIN {X 0.053,Y -220.318,Z 1288.176,A 0.000,B 0.000,C 90.000,E1 31.671} C_DIS
LIN {X -0.130,Y -215.274,Z 1288.155,A 0.000,B 0.000,C 90.000,E1 27.847} C_DIS
LIN {X 0.000,Y -210.762,Z 1288.133,A 0.000,B 0.000,C 90.000,E1 23.898} C_DIS
LIN {X 0.030,Y -206.842,Z 1288.111,A 0.000,B 0.000,C 90.000,E1 19.939} C_DIS
LIN {X -0.093,Y -202.727,Z 1288.084,A 0.000,B 0.000,C 90.000,E1 15.190} C_DIS
LIN {X -0.089,Y -199.100,Z 1288.053,A 0.000,B 0.000,C 90.000,E1 9.557} C_DIS
LIN {X -0.012,Y -196.511,Z 1288.012,A 0.000,B 0.000,C 90.000,E1 2.236} C_DIS
LIN {X 0.050,Y -198.089,Z 1287.948,A 0.000,B 0.000,C 90.000,E1 350.566} C_DIS
LIN {X -0.072,Y -201.691,Z 1287.916,A 0.000,B 0.000,C 90.000,E1 344.936} C_DIS
LIN {X -0.057,Y -205.874,Z 1287.889,A 0.000,B 0.000,C 90.000,E1 340.115} C_DIS
LIN {X 0.069,Y -210.233,Z 1287.867,A 0.000,B 0.000,C 90.000,E1 336.102} C_DIS
LIN {X 0.099,Y -215.319,Z 1287.845,A 0.000,B 0.000,C 90.000,E1 332.153} C_DIS
LIN {X 0.014,Y -221.175,Z 1287.824,A 0.000,B 0.000,C 90.000,E1 328.280} C_DIS
LIN {X 0.136,Y -227.852,Z 1287.802,A 0.000,B 0.000,C 90.000,E1 324.402} C_DIS
LIN {X 0.009,Y -235.491,Z 1287.781,A 0.000,B 0.000,C 90.000,E1 320.642} C_DIS
LIN {X 0.030,Y -244.100,Z 1287.761,A 0.000,B 0.000,C 90.000,E1 316.905} C_DIS
LIN {X -0.049,Y -252.955,Z 1287.742,A 0.000,B 0.000,C 90.000,E1 313.623} C_DIS
LIN {X 0.056,Y -259.606,Z 1287.730,A 0.000,B 0.000,C 90.000,E1 311.434} C_DIS
LIN {X 0.006,Y -268.401,Z 1287.716,A 0.000,B 0.000,C 90.000,E1 308.955} C_DIS
LIN {X 0.035,Y -278.527,Z 1287.703,A 0.000,B 0.000,C 90.000,E1 306.503} C_DIS
LIN {X -0.134,Y -286.601,Z 1287.693,A 0.000,B 0.000,C 90.000,E1 304.818} C_DIS
LIN {X 0.068,Y -295.459,Z 1287.684,A 0.000,B 0.000,C 90.000,E1 303.086} C_DIS
LIN {X -0.166,Y -305.166,Z 1287.675,A 0.000,B 0.000,C 90.000,E1 301.465} C_DIS
LIN {X -0.033,Y -313.717,Z 1287.667,A 0.000,B 0.000,C 90.000,E1 300.129} C_DIS
LIN {X -0.118,Y -330.223,Z 1287.655,A 0.000,B 0.000,C 90.000,E1 297.897} C_DIS
LIN {X -0.008,Y -350.457,Z 1287.641,A 0.000,B 0.000,C 90.000,E1 295.412} C_DIS
LIN {X 0.043,Y -363.530,Z 1287.633,A 0.000,B 0.000,C 90.000,E1 293.898} C_DIS
LIN {X 0.048,Y -373.747,Z 1287.626,A 0.000,B 0.000,C 90.000,E1 292.717} C_DIS
LIN {X -0.066,Y -386.195,Z 1287.618,A 0.000,B 0.000,C 90.000,E1 291.280} C_DIS
LIN {X 0.237,Y -410.984,Z 1287.603,A 0.000,B 0.000,C 90.000,E1 288.417} C_DIS
LIN {X 0.075,Y -420.978,Z 1287.596,A 0.000,B 0.000,C 90.000,E1 287.347} C_DIS
LIN {X 0.084,Y -430.489,Z 1287.590,A 0.000,B 0.000,C 90.000,E1 286.260} C_DIS
LIN {X -0.111,Y -437.113,Z 1287.586,A 0.000,B 0.000,C 90.000,E1 285.481} C_DIS
LIN {X 0.063,Y -443.001,Z 1287.582,A 0.000,B 0.000,C 90.000,E1 284.662} C_DIS
LIN {X -0.029,Y -448.187,Z 1287.577,A 0.000,B 0.000,C 90.000,E1 283.883} C_DIS
LIN {X -0.183,Y -452.714,Z 1287.573,A 0.000,B 0.000,C 90.000,E1 283.119} C_DIS
LIN {X 0.143,Y -456.655,Z 1287.568,A 0.000,B 0.000,C 90.000,E1 282.299} C_DIS
LIN {X 0.235,Y -458.922,Z 1287.566,A 0.000,B 0.000,C 90.000,E1 281.771} C_DIS
LIN {X -0.110,Y -460.931,Z 1287.563,A 0.000,B 0.000,C 90.000,E1 281.299} C_DIS
LIN {X -0.087,Y -462.627,Z 1287.560,A 0.000,B 0.000,C 90.000,E1 280.782} C_DIS
LIN {X 0.036,Y -464.028,Z 1287.557,A 0.000,B 0.000,C 90.000,E1 280.254} C_DIS
LIN {X 0.166,Y -465.070,Z 1287.554,A 0.000,B 0.000,C 90.000,E1 279.726} C_DIS
LIN {X 0.227,Y -465.695,Z 1287.551,A 0.000,B 0.000,C 90.000,E1 279.208} C_DIS
LIN {X -0.163,Y -466.005,Z 1287.548,A 0.000,B 0.000,C 90.000,E1 278.746} C_DIS
LIN {X -0.021,Y -465.881,Z 1287.546,A 0.000,B 0.000,C 90.000,E1 278.219} C_DIS
LIN {X 0.056,Y -465.209,Z 1287.543,A 0.000,B 0.000,C 90.000,E1 277.701} C_DIS
LIN {X 0.133,Y -464.129,Z 1287.540,A 0.000,B 0.000,C 90.000,E1 277.182} C_DIS
LIN {X 0.207,Y -462.528,Z 1287.537,A 0.000,B 0.000,C 90.000,E1 276.663} C_DIS
LIN {X -0.184,Y -460.513,Z 1287.534,A 0.000,B 0.000,C 90.000,E1 276.201} C_DIS
LIN {X 0.144,Y -456.796,Z 1287.530,A 0.000,B 0.000,C 90.000,E1 275.391} C_DIS
LIN {X 0.133,Y -453.849,Z 1287.527,A 0.000,B 0.000,C 90.000,E1 274.878} C_DIS
LIN {X 0.146,Y -450.189,Z 1287.524,A 0.000,B 0.000,C 90.000,E1 274.359} C_DIS
LIN {X 0.138,Y -445.662,Z 1287.521,A 0.000,B 0.000,C 90.000,E1 273.841} C_DIS
LIN {X 0.213,Y -440.113,Z 1287.519,A 0.000,B 0.000,C 90.000,E1 273.326} C_DIS
LIN {X 0.199,Y -433.963,Z 1287.516,A 0.000,B 0.000,C 90.000,E1 272.865} C_DIS
LIN {X 0.176,Y -427.299,Z 1287.514,A 0.000,B 0.000,C 90.000,E1 272.465} C_DIS
LIN {X 0.199,Y -420.377,Z 1287.512,A 0.000,B 0.000,C 90.000,E1 272.121} C_DIS
LIN {X -0.179,Y -413.302,Z 1287.510,A 0.000,B 0.000,C 90.000,E1 271.892} C_DIS
LIN {X -0.192,Y -406.274,Z 1287.509,A 0.000,B 0.000,C 90.000,E1 271.661} C_DIS
LIN {X 0.053,Y -399.195,Z 1287.508,A 0.000,B 0.000,C 90.000,E1 271.432} C_DIS
LIN {X 0.120,Y -391.807,Z 1287.507,A 0.000,B 0.000,C 90.000,E1 271.260} C_DIS
LIN {X -0.006,Y -383.474,Z 1287.506,A 0.000,B 0.000,C 90.000,E1 271.146} C_DIS
LIN {X -0.101,Y -370.982,Z 1287.506,A 0.000,B 0.000,C 90.000,E1 271.031} C_DIS
LIN {X -0.038,Y -359.202,Z 1287.505,A 0.000,B 0.000,C 90.000,E1 270.974} C_DIS
LIN {X -0.044,Y -181.464,Z 1287.505,A 0.000,B 0.000,C 90.000,E1 270.974} C_DIS
LIN {X 0.089,Y -181.572,Z 1287.500,A 0.000,B 0.000,C 90.000,E1 270.057} C_DIS
LIN {X 0.076,Y -180.868,Z 1287.472,A 0.000,B 0.000,C 90.000,E1 265.008} C_DIS
LIN {X -0.047,Y -178.984,Z 1287.444,A 0.000,B 0.000,C 90.000,E1 259.982} C_DIS
LIN {X -0.036,Y -177.960,Z 1287.435,A 0.000,B 0.000,C 90.000,E1 258.285} C_DIS
LIN {X -0.016,Y -175.602,Z 1287.411,A 0.000,B 0.000,C 90.000,E1 254.031} C_DIS
LIN {X -0.004,Y -172.325,Z 1287.387,A 0.000,B 0.000,C 90.000,E1 249.752} C_DIS
LIN {X -0.025,Y -171.803,Z 1287.383,A 0.000,B 0.000,C 90.000,E1 248.901} C_DIS
LIN {X 0.012,Y -169.478,Z 1287.368,A 0.000,B 0.000,C 90.000,E1 246.305} C_DIS
LIN {X -0.081,Y -166.804,Z 1287.349,A 0.000,B 0.000,C 90.000,E1 242.871} C_DIS
LIN {X 0.062,Y -162.785,Z 1287.325,A 0.000,B 0.000,C 90.000,E1 238.456} C_DIS
LIN {X 0.038,Y -161.473,Z 1287.315,A 0.000,B 0.000,C 90.000,E1 236.707} C_DIS
LIN {X 0.078,Y -157.468,Z 1287.291,A 0.000,B 0.000,C 90.000,E1 232.271} C_DIS
LIN {X 0.011,Y -155.482,Z 1287.276,A 0.000,B 0.000,C 90.000,E1 229.622} C_DIS
LIN {X -0.057,Y -151.792,Z 1287.251,A 0.000,B 0.000,C 90.000,E1 225.162} C_DIS
LIN {X -0.043,Y -149.999,Z 1287.236,A 0.000,B 0.000,C 90.000,E1 222.447} C_DIS
LIN {X -0.012,Y -146.828,Z 1287.210,A 0.000,B 0.000,C 90.000,E1 217.890} C_DIS
LIN {X -0.025,Y -145.408,Z 1287.195,A 0.000,B 0.000,C 90.000,E1 215.152} C_DIS
LIN {X 0.011,Y -142.839,Z 1287.170,A 0.000,B 0.000,C 90.000,E1 210.541} C_DIS
LIN {X -0.059,Y -141.453,Z 1287.149,A 0.000,B 0.000,C 90.000,E1 206.873} C_DIS
LIN {X -0.020,Y -139.372,Z 1287.113,A 0.000,B 0.000,C 90.000,E1 200.355} C_DIS
LIN {X -0.077,Y -138.822,Z 1287.098,A 0.000,B 0.000,C 90.000,E1 197.583} C_DIS
LIN {X 0.011,Y -138.352,Z 1287.056,A 0.000,B 0.000,C 90.000,E1 190.074} C_DIS
LIN {X -0.016,Y -139.533,Z 1287.004,A 0.000,B 0.000,C 90.000,E1 180.745} C_DIS
LIN {X -0.064,Y -141.216,Z 1286.973,A 0.000,B 0.000,C 90.000,E1 175.179} C_DIS
LIN {X 0.037,Y -142.590,Z 1286.958,A 0.000,B 0.000,C 90.000,E1 172.356} C_DIS
LIN {X -0.010,Y -144.889,Z 1286.932,A 0.000,B 0.000,C 90.000,E1 167.757} C_DIS
LIN {X -0.056,Y -147.517,Z 1286.911,A 0.000,B 0.000,C 90.000,E1 164.102} C_DIS
LIN {X 0.018,Y -150.112,Z 1286.891,A 0.000,B 0.000,C 90.000,E1 160.423} C_DIS
LIN {X 0.030,Y -153.471,Z 1286.871,A 0.000,B 0.000,C 90.000,E1 156.794} C_DIS
LIN {X 0.021,Y -157.835,Z 1286.846,A 0.000,B 0.000,C 90.000,E1 152.308} C_DIS
LIN {X 0.051,Y -162.119,Z 1286.826,A 0.000,B 0.000,C 90.000,E1 148.742} C_DIS
LIN {X -0.064,Y -166.321,Z 1286.807,A 0.000,B 0.000,C 90.000,E1 145.261} C_DIS
LIN {X 0.038,Y -171.339,Z 1286.787,A 0.000,B 0.000,C 90.000,E1 141.743} C_DIS
LIN {X -0.035,Y -176.242,Z 1286.768,A 0.000,B 0.000,C 90.000,E1 138.324} C_DIS
LIN {X 0.084,Y -180.522,Z 1286.754,A 0.000,B 0.000,C 90.000,E1 135.729} C_DIS
LIN {X 0.064,Y -185.925,Z 1286.735,A 0.000,B 0.000,C 90.000,E1 132.366} C_DIS
LIN {X -0.001,Y -190.554,Z 1286.722,A 0.000,B 0.000,C 90.000,E1 129.886} C_DIS
LIN {X 0.030,Y -196.305,Z 1286.703,A 0.000,B 0.000,C 90.000,E1 126.583} C_DIS
LIN {X 0.080,Y -199.765,Z 1286.694,A 0.000,B 0.000,C 90.000,E1 124.818} C_DIS
LIN {X 0.073,Y -309.773,Z 1286.693,A 0.000,B 0.000,C 90.000,E1 124.818} C_DIS
LIN {X 0.013,Y -314.702,Z 1286.693,A 0.000,B 0.000,C 90.000,E1 124.659} C_DIS
LIN {X 0.033,Y -317.094,Z 1286.692,A 0.000,B 0.000,C 90.000,E1 124.485} C_DIS
LIN {X 0.172,Y -320.313,Z 1286.690,A 0.000,B 0.000,C 90.000,E1 124.119} C_DIS
LIN {X -0.039,Y -322.286,Z 1286.688,A 0.000,B 0.000,C 90.000,E1 123.865} C_DIS
LIN {X -0.072,Y -323.829,Z 1286.687,A 0.000,B 0.000,C 90.000,E1 123.579} C_DIS
LIN {X -0.165,Y -326.266,Z 1286.683,A 0.000,B 0.000,C 90.000,E1 122.959} C_DIS
LIN {X -0.160,Y -336.851,Z 1286.667,A 0.000,B 0.000,C 90.000,E1 120.129} C_DIS
LIN {X -0.062,Y -348.792,Z 1286.652,A 0.000,B 0.000,C 90.000,E1 117.334} C_DIS
LIN {X 0.082,Y -362.189,Z 1286.637,A 0.000,B 0.000,C 90.000,E1 114.591} C_DIS
LIN {X 0.203,Y -375.417,Z 1286.624,A 0.000,B 0.000,C 90.000,E1 112.206} C_DIS
LIN {X -0.131,Y -389.983,Z 1286.611,A 0.000,B 0.000,C 90.000,E1 109.939} C_DIS
LIN {X 0.134,Y -405.985,Z 1286.598,A 0.000,B 0.000,C 90.000,E1 107.638} C_DIS
LIN {X 0.170,Y -423.540,Z 1286.586,A 0.000,B 0.000,C 90.000,E1 105.426} C_DIS
LIN {X 0.030,Y -442.735,Z 1286.574,A 0.000,B 0.000,C 90.000,E1 103.300} C_DIS
LIN {X 0.019,Y -462.848,Z 1286.563,A 0.000,B 0.000,C 90.000,E1 101.299} C_DIS
LIN {X -0.070,Y -475.709,Z 1286.556,A 0.000,B 0.000,C 90.000,E1 100.141} C_DIS
LIN {X 0.018,Y -477.933,Z 1286.555,A 0.000,B 0.000,C 90.000,E1 99.905} C_DIS
LIN {X 0.106,Y -479.617,Z 1286.554,A 0.000,B 0.000,C 90.000,E1 99.670} C_DIS
LIN {X -0.098,Y -481.044,Z 1286.552,A 0.000,B 0.000,C 90.000,E1 99.443} C_DIS
LIN {X -0.224,Y -482.106,Z 1286.551,A 0.000,B 0.000,C 90.000,E1 99.208} C_DIS
LIN {X 0.014,Y -483.340,Z 1286.548,A 0.000,B 0.000,C 90.000,E1 98.681} C_DIS
LIN {X 0.186,Y -483.557,Z 1286.545,A 0.000,B 0.000,C 90.000,E1 98.163} C_DIS
LIN {X -0.112,Y -482.794,Z 1286.543,A 0.000,B 0.000,C 90.000,E1 97.701} C_DIS
LIN {X 0.071,Y -480.925,Z 1286.540,A 0.000,B 0.000,C 90.000,E1 97.182} C_DIS
LIN {X -0.049,Y -479.463,Z 1286.539,A 0.000,B 0.000,C 90.000,E1 96.947} C_DIS
LIN {X 0.181,Y -466.446,Z 1286.529,A 0.000,B 0.000,C 90.000,E1 95.163} C_DIS
LIN {X 0.126,Y -450.758,Z 1286.516,A 0.000,B 0.000,C 90.000,E1 92.865} C_DIS
LIN {X -0.088,Y -437.466,Z 1286.504,A 0.000,B 0.000,C 90.000,E1 90.802} C_DIS
LIN {X 0.026,Y -418.065,Z 1286.485,A 0.000,B 0.000,C 90.000,E1 87.306} C_DIS
LIN {X -0.128,Y -407.911,Z 1286.474,A 0.000,B 0.000,C 90.000,E1 85.412} C_DIS
LIN {X -0.008,Y -397.770,Z 1286.464,A 0.000,B 0.000,C 90.000,E1 83.451} C_DIS
LIN {X -0.100,Y -387.462,Z 1286.453,A 0.000,B 0.000,C 90.000,E1 81.489} C_DIS
LIN {X 0.060,Y -378.299,Z 1286.443,A 0.000,B 0.000,C 90.000,E1 79.746} C_DIS
LIN {X 0.119,Y -368.816,Z 1286.433,A 0.000,B 0.000,C 90.000,E1 77.993} C_DIS
LIN {X 0.084,Y -359.032,Z 1286.424,A 0.000,B 0.000,C 90.000,E1 76.228} C_DIS
LIN {X -0.036,Y -349.131,Z 1286.414,A 0.000,B 0.000,C 90.000,E1 74.448} C_DIS
LIN {X -0.007,Y -337.551,Z 1286.402,A 0.000,B 0.000,C 90.000,E1 72.308} C_DIS
LIN {X -0.112,Y -323.011,Z 1286.386,A 0.000,B 0.000,C 90.000,E1 69.518} C_DIS
LIN {X -0.014,Y -306.398,Z 1286.366,A 0.000,B 0.000,C 90.000,E1 65.973} C_DIS
LIN {X 0.044,Y -295.453,Z 1286.352,A 0.000,B 0.000,C 90.000,E1 63.332} C_DIS
LIN {X 0.138,Y -288.124,Z 1286.341,A 0.000,B 0.000,C 90.000,E1 61.307} C_DIS
LIN {X 0.029,Y -279.347,Z 1286.326,A 0.000,B 0.000,C 90.000,E1 58.614} C_DIS
LIN {X -0.055,Y -269.461,Z 1286.307,A 0.000,B 0.000,C 90.000,E1 55.182} C_DIS
LIN {X -0.031,Y -260.288,Z 1286.287,A 0.000,B 0.000,C 90.000,E1 51.662} C_DIS
LIN {X 0.126,Y -253.273,Z 1286.271,A 0.000,B 0.000,C 90.000,E1 48.771} C_DIS
LIN {X 0.054,Y -246.507,Z 1286.255,A 0.000,B 0.000,C 90.000,E1 45.891} C_DIS
LIN {X -0.055,Y -238.459,Z 1286.235,A 0.000,B 0.000,C 90.000,E1 42.243} C_DIS
LIN {X 0.133,Y -231.125,Z 1286.214,A 0.000,B 0.000,C 90.000,E1 38.463} C_DIS
LIN {X 0.062,Y -224.673,Z 1286.193,A 0.000,B 0.000,C 90.000,E1 34.692} C_DIS
LIN {X -0.026,Y -218.967,Z 1286.172,A 0.000,B 0.000,C 90.000,E1 30.875} C_DIS
LIN {X -0.060,Y -213.999,Z 1286.150,A 0.000,B 0.000,C 90.000,E1 27.001} C_DIS
LIN {X -0.035,Y -208.782,Z 1286.124,A 0.000,B 0.000,C 90.000,E1 22.280} C_DIS
LIN {X -0.017,Y -204.998,Z 1286.102,A 0.000,B 0.000,C 90.000,E1 18.308} C_DIS
LIN {X 0.071,Y -201.171,Z 1286.075,A 0.000,B 0.000,C 90.000,E1 13.480} C_DIS
LIN {X -0.072,Y -197.959,Z 1286.044,A 0.000,B 0.000,C 90.000,E1 7.871} C_DIS
LIN {X -0.036,Y -195.926,Z 1285.997,A 0.000,B 0.000,C 90.000,E1 359.542} C_DIS
LIN {X 0.034,Y -197.939,Z 1285.948,A 0.000,B 0.000,C 90.000,E1 350.566} C_DIS
LIN {X -0.093,Y -201.603,Z 1285.916,A 0.000,B 0.000,C 90.000,E1 344.936} C_DIS
LIN {X 0.112,Y -205.833,Z 1285.889,A 0.000,B 0.000,C 90.000,E1 340.061} C_DIS
LIN {X 0.043,Y -210.228,Z 1285.867,A 0.000,B 0.000,C 90.000,E1 336.102} C_DIS
LIN {X 0.074,Y -215.331,Z 1285.845,A 0.000,B 0.000,C 90.000,E1 332.153} C_DIS
LIN {X -0.012,Y -221.178,Z 1285.824,A 0.000,B 0.000,C 90.000,E1 328.280} C_DIS
LIN {X 0.109,Y -227.883,Z 1285.802,A 0.000,B 0.000,C 90.000,E1 324.402} C_DIS
LIN {X -0.019,Y -235.524,Z 1285.781,A 0.000,B 0.000,C 90.000,E1 320.642} C_DIS
LIN {X 0.003,Y -244.120,Z 1285.761,A 0.000,B 0.000,C 90.000,E1 316.905} C_DIS
LIN {X -0.068,Y -254.006,Z 1285.740,A 0.000,B 0.000,C 90.000,E1 313.257} C_DIS
LIN {X 0.064,Y -260.783,Z 1285.728,A 0.000,B 0.000,C 90.000,E1 311.067} C_DIS
LIN {X -0.024,Y -268.377,Z 1285.716,A 0.000,B 0.000,C 90.000,E1 308.955} C_DIS
LIN {X 0.004,Y -278.506,Z 1285.703,A 0.000,B 0.000,C 90.000,E1 306.503} C_DIS
LIN {X 0.069,Y -286.580,Z 1285.693,A 0.000,B 0.000,C 90.000,E1 304.771} C_DIS
LIN {X 0.035,Y -295.432,Z 1285.684,A 0.000,B 0.000,C 90.000,E1 303.086} C_DIS
LIN {X 0.059,Y -305.122,Z 1285.675,A 0.000,B 0.000,C 90.000,E1 301.416} C_DIS
LIN {X -0.070,Y -313.684,Z 1285.667,A 0.000,B 0.000,C 90.000,E1 300.129} C_DIS
LIN {X 0.134,Y -330.194,Z 1285.655,A 0.000,B 0.000,C 90.000,E1 297.847} C_DIS
LIN {X -0.037,Y -350.387,Z 1285.641,A 0.000,B 0.000,C 90.000,E1 295.412} C_DIS
LIN {X 0.006,Y -363.467,Z 1285.633,A 0.000,B 0.000,C 90.000,E1 293.898} C_DIS
LIN {X 0.090,Y -376.273,Z 1285.625,A 0.000,B 0.000,C 90.000,E1 292.408} C_DIS
LIN {X -0.011,Y -388.666,Z 1285.616,A 0.000,B 0.000,C 90.000,E1 290.972} C_DIS
LIN {X -0.121,Y -415.983,Z 1285.599,A 0.000,B 0.000,C 90.000,E1 287.928} C_DIS
LIN {X 0.136,Y -425.738,Z 1285.594,A 0.000,B 0.000,C 90.000,E1 286.804} C_DIS
LIN {X 0.079,Y -434.899,Z 1285.587,A 0.000,B 0.000,C 90.000,E1 285.733} C_DIS
LIN {X -0.080,Y -441.061,Z 1285.583,A 0.000,B 0.000,C 90.000,E1 284.954} C_DIS
LIN {X 0.247,Y -446.536,Z 1285.579,A 0.000,B 0.000,C 90.000,E1 284.120} C_DIS
LIN {X 0.075,Y -451.284,Z 1285.574,A 0.000,B 0.000,C 90.000,E1 283.355} C_DIS
LIN {X -0.049,Y -455.454,Z 1285.570,A 0.000,B 0.000,C 90.000,E1 282.591} C_DIS
LIN {X -0.144,Y -459.011,Z 1285.566,A 0.000,B 0.000,C 90.000,E1 281.827} C_DIS
LIN {X -0.040,Y -461.002,Z 1285.563,A 0.000,B 0.000,C 90.000,E1 281.299} C_DIS
LIN {X -0.016,Y -462.709,Z 1285.560,A 0.000,B 0.000,C 90.000,E1 280.782} C_DIS
LIN {X 0.107,Y -464.100,Z 1285.557,A 0.000,B 0.000,C 90.000,E1 280.254} C_DIS
LIN {X 0.238,Y -465.201,Z 1285.554,A 0.000,B 0.000,C 90.000,E1 279.726} C_DIS
LIN {X -0.160,Y -465.864,Z 1285.551,A 0.000,B 0.000,C 90.000,E1 279.265} C_DIS
LIN {X -0.090,Y -466.146,Z 1285.549,A 0.000,B 0.000,C 90.000,E1 278.746} C_DIS
LIN {X 0.054,Y -466.034,Z 1285.546,A 0.000,B 0.000,C 90.000,E1 278.219} C_DIS
LIN {X 0.131,Y -465.426,Z 1285.543,A 0.000,B 0.000,C 90.000,E1 277.701} C_DIS
LIN {X 0.208,Y -464.353,Z 1285.540,A 0.000,B 0.000,C 90.000,E1 277.182} C_DIS
LIN {X -0.176,Y -462.817,Z 1285.537,A 0.000,B 0.000,C 90.000,E1 276.720} C_DIS
LIN {X 0.176,Y -459.686,Z 1285.533,A 0.000,B 0.000,C 90.000,E1 275.910} C_DIS
LIN {X 0.224,Y -457.216,Z 1285.530,A 0.000,B 0.000,C 90.000,E1 275.391} C_DIS
LIN {X -0.239,Y -454.306,Z 1285.527,A 0.000,B 0.000,C 90.000,E1 274.935} C_DIS
LIN {X -0.219,Y -450.736,Z 1285.524,A 0.000,B 0.000,C 90.000,E1 274.416} C_DIS
LIN {X 0.225,Y -446.272,Z 1285.521,A 0.000,B 0.000,C 90.000,E1 273.841} C_DIS
LIN {X -0.182,Y -440.848,Z 1285.519,A 0.000,B 0.000,C 90.000,E1 273.383} C_DIS
LIN {X 0.216,Y -434.674,Z 1285.516,A 0.000,B 0.000,C 90.000,E1 272.865} C_DIS
LIN {X 0.198,Y -428.159,Z 1285.514,A 0.000,B 0.000,C 90.000,E1 272.465} C_DIS
LIN {X -0.207,Y -421.302,Z 1285.512,A 0.000,B 0.000,C 90.000,E1 272.178} C_DIS
LIN {X -0.181,Y -414.279,Z 1285.510,A 0.000,B 0.000,C 90.000,E1 271.892} C_DIS
LIN {X 0.185,Y -407.195,Z 1285.509,A 0.000,B 0.000,C 90.000,E1 271.604} C_DIS
LIN {X -0.009,Y -400.158,Z 1285.508,A 0.000,B 0.000,C 90.000,E1 271.432} C_DIS
LIN {X 0.029,Y -392.805,Z 1285.507,A 0.000,B 0.000,C 90.000,E1 271.260} C_DIS
LIN {X -0.110,Y -384.550,Z 1285.506,A 0.000,B 0.000,C 90.000,E1 271.146} C_DIS
LIN {X -0.054,Y -375.233,Z 1285.506,A 0.000,B 0.000,C 90.000,E1 271.031} C_DIS
LIN {X -0.150,Y -363.352,Z 1285.505,A 0.000,B 0.000,C 90.000,E1 270.974} C_DIS
LIN {X 0.156,Y -358.065,Z 1285.505,A 0.000,B 0.000,C 90.000,E1 270.917} C_DIS
LIN {X 0.051,Y -181.471,Z 1285.505,A 0.000,B 0.000,C 90.000,E1 270.917} C_DIS
LIN {X 0.043,Y -181.542,Z 1285.499,A 0.000,B 0.000,C 90.000,E1 269.885} C_DIS
LIN {X -0.014,Y -180.907,Z 1285.475,A 0.000,B 0.000,C 90.000,E1 265.527} C_DIS
LIN {X 0.043,Y -180.759,Z 1285.470,A 0.000,B 0.000,C 90.000,E1 264.666} C_DIS
LIN {X -0.064,Y -178.852,Z 1285.442,A 0.000,B 0.000,C 90.000,E1 259.634} C_DIS
LIN {X 0.007,Y -175.896,Z 1285.414,A 0.000,B 0.000,C 90.000,E1 254.519} C_DIS
LIN {X -0.054,Y -174.570,Z 1285.405,A 0.000,B 0.000,C 90.000,E1 252.834} C_DIS
LIN {X -0.018,Y -171.554,Z 1285.381,A 0.000,B 0.000,C 90.000,E1 248.539} C_DIS
LIN {X 0.037,Y -167.778,Z 1285.357,A 0.000,B 0.000,C 90.000,E1 244.204} C_DIS
LIN {X -0.021,Y -166.490,Z 1285.347,A 0.000,B 0.000,C 90.000,E1 242.487} C_DIS
LIN {X -0.025,Y -163.201,Z 1285.328,A 0.000,B 0.000,C 90.000,E1 238.997} C_DIS
LIN {X 0.030,Y -161.165,Z 1285.313,A 0.000,B 0.000,C 90.000,E1 236.342} C_DIS
LIN {X 0.064,Y -157.180,Z 1285.288,A 0.000,B 0.000,C 90.000,E1 231.904} C_DIS
LIN {X -0.013,Y -155.910,Z 1285.279,A 0.000,B 0.000,C 90.000,E1 230.150} C_DIS
LIN {X 0.044,Y -152.161,Z 1285.254,A 0.000,B 0.000,C 90.000,E1 225.648} C_DIS
LIN {X 0.063,Y -150.409,Z 1285.239,A 0.000,B 0.000,C 90.000,E1 222.933} C_DIS
LIN {X 0.086,Y -147.139,Z 1285.213,A 0.000,B 0.000,C 90.000,E1 218.382} C_DIS
LIN {X -0.008,Y -145.698,Z 1285.198,A 0.000,B 0.000,C 90.000,E1 215.678} C_DIS
LIN {X 0.000,Y -143.081,Z 1285.173,A 0.000,B 0.000,C 90.000,E1 211.082} C_DIS
LIN {X 0.005,Y -141.700,Z 1285.152,A 0.000,B 0.000,C 90.000,E1 207.385} C_DIS
LIN {X -0.072,Y -139.465,Z 1285.116,A 0.000,B 0.000,C 90.000,E1 200.918} C_DIS
LIN {X -0.018,Y -139.199,Z 1285.106,A 0.000,B 0.000,C 90.000,E1 199.033} C_DIS
LIN {X 0.046,Y -138.327,Z 1285.054,A 0.000,B 0.000,C 90.000,E1 189.670} C_DIS
LIN {X 0.050,Y -139.446,Z 1285.007,A 0.000,B 0.000,C 90.000,E1 181.260} C_DIS
LIN {X -0.009,Y -140.985,Z 1284.976,A 0.000,B 0.000,C 90.000,E1 175.698} C_DIS
LIN {X -0.060,Y -142.740,Z 1284.955,A 0.000,B 0.000,C 90.000,E1 172.008} C_DIS
LIN {X 0.038,Y -145.133,Z 1284.930,A 0.000,B 0.000,C 90.000,E1 167.353} C_DIS
LIN {X 0.032,Y -147.756,Z 1284.909,A 0.000,B 0.000,C 90.000,E1 163.685} C_DIS
LIN {X -0.029,Y -150.427,Z 1284.889,A 0.000,B 0.000,C 90.000,E1 160.061} C_DIS
LIN {X -0.014,Y -153.869,Z 1284.869,A 0.000,B 0.000,C 90.000,E1 156.433} C_DIS
LIN {X 0.042,Y -157.280,Z 1284.849,A 0.000,B 0.000,C 90.000,E1 152.820} C_DIS
LIN {X -0.020,Y -161.459,Z 1284.829,A 0.000,B 0.000,C 90.000,E1 149.282} C_DIS
LIN {X -0.014,Y -165.659,Z 1284.810,A 0.000,B 0.000,C 90.000,E1 145.754} C_DIS
LIN {X -0.032,Y -170.595,Z 1284.790,A 0.000,B 0.000,C 90.000,E1 142.271} C_DIS
LIN {X 0.007,Y -175.473,Z 1284.771,A 0.000,B 0.000,C 90.000,E1 138.809} C_DIS
LIN {X -0.011,Y -181.094,Z 1284.752,A 0.000,B 0.000,C 90.000,E1 135.405} C_DIS
LIN {X -0.021,Y -186.538,Z 1284.734,A 0.000,B 0.000,C 90.000,E1 132.043} C_DIS
LIN {X -0.080,Y -191.154,Z 1284.720,A 0.000,B 0.000,C 90.000,E1 129.564} C_DIS
LIN {X -0.002,Y -196.957,Z 1284.701,A 0.000,B 0.000,C 90.000,E1 126.251} C_DIS
LIN {X 0.051,Y -199.782,Z 1284.693,A 0.000,B 0.000,C 90.000,E1 124.818} C_DIS
LIN {X 0.042,Y -308.739,Z 1284.693,A 0.000,B 0.000,C 90.000,E1 124.818} C_DIS
LIN {X -0.081,Y -313.248,Z 1284.693,A 0.000,B 0.000,C 90.000,E1 124.739} C_DIS
LIN {X 0.054,Y -315.168,Z 1284.692,A 0.000,B 0.000,C 90.000,E1 124.612} C_DIS
LIN {X 0.089,Y -319.017,Z 1284.691,A 0.000,B 0.000,C 90.000,E1 124.278} C_DIS
LIN {X 0.093,Y -322.561,Z 1284.688,A 0.000,B 0.000,C 90.000,E1 123.785} C_DIS
LIN {X -0.099,Y -324.178,Z 1284.686,A 0.000,B 0.000,C 90.000,E1 123.499} C_DIS
LIN {X -0.102,Y -327.660,Z 1284.681,A 0.000,B 0.000,C 90.000,E1 122.546} C_DIS
LIN {X -0.060,Y -338.429,Z 1284.665,A 0.000,B 0.000,C 90.000,E1 119.716} C_DIS
LIN {X 0.080,Y -350.570,Z 1284.650,A 0.000,B 0.000,C 90.000,E1 116.924} C_DIS
LIN {X 0.114,Y -364.181,Z 1284.635,A 0.000,B 0.000,C 90.000,E1 114.207} C_DIS
LIN {X 0.140,Y -377.615,Z 1284.621,A 0.000,B 0.000,C 90.000,E1 111.844} C_DIS
LIN {X -0.137,Y -392.400,Z 1284.609,A 0.000,B 0.000,C 90.000,E1 109.577} C_DIS
LIN {X 0.190,Y -408.642,Z 1284.596,A 0.000,B 0.000,C 90.000,E1 107.275} C_DIS
LIN {X -0.231,Y -426.454,Z 1284.584,A 0.000,B 0.000,C 90.000,E1 105.134} C_DIS
LIN {X -0.258,Y -445.857,Z 1284.572,A 0.000,B 0.000,C 90.000,E1 103.008} C_DIS
LIN {X -0.063,Y -466.061,Z 1284.561,A 0.000,B 0.000,C 90.000,E1 101.007} C_DIS
LIN {X -0.017,Y -476.331,Z 1284.556,A 0.000,B 0.000,C 90.000,E1 100.074} C_DIS
LIN {X -0.026,Y -478.378,Z 1284.555,A 0.000,B 0.000,C 90.000,E1 99.849} C_DIS
LIN {X -0.156,Y -480.083,Z 1284.553,A 0.000,B 0.000,C 90.000,E1 99.613} C_DIS
LIN {X 0.189,Y -481.362,Z 1284.552,A 0.000,B 0.000,C 90.000,E1 99.321} C_DIS
LIN {X -0.129,Y -482.943,Z 1284.549,A 0.000,B 0.000,C 90.000,E1 98.859} C_DIS
LIN {X 0.040,Y -483.461,Z 1284.546,A 0.000,B 0.000,C 90.000,E1 98.341} C_DIS
LIN {X -0.192,Y -483.002,Z 1284.544,A 0.000,B 0.000,C 90.000,E1 97.871} C_DIS
LIN {X -0.011,Y -481.499,Z 1284.541,A 0.000,B 0.000,C 90.000,E1 97.352} C_DIS
LIN {X -0.190,Y -480.275,Z 1284.539,A 0.000,B 0.000,C 90.000,E1 97.125} C_DIS
LIN {X 0.167,Y -478.643,Z 1284.538,A 0.000,B 0.000,C 90.000,E1 96.834} C_DIS
LIN {X -0.092,Y -465.633,Z 1284.528,A 0.000,B 0.000,C 90.000,E1 95.106} C_DIS
LIN {X -0.152,Y -449.950,Z 1284.516,A 0.000,B 0.000,C 90.000,E1 92.808} C_DIS
LIN {X 0.061,Y -436.699,Z 1284.504,A 0.000,B 0.000,C 90.000,E1 90.688} C_DIS
LIN {X 0.136,Y -417.339,Z 1284.484,A 0.000,B 0.000,C 90.000,E1 87.192} C_DIS
LIN {X 0.063,Y -405.736,Z 1284.472,A 0.000,B 0.000,C 90.000,E1 85.008} C_DIS
LIN {X 0.063,Y -397.050,Z 1284.463,A 0.000,B 0.000,C 90.000,E1 83.337} C_DIS
LIN {X -0.046,Y -386.724,Z 1284.452,A 0.000,B 0.000,C 90.000,E1 81.376} C_DIS
LIN {X 0.096,Y -377.560,Z 1284.443,A 0.000,B 0.000,C 90.000,E1 79.634} C_DIS
LIN {X 0.140,Y -369.660,Z 1284.434,A 0.000,B 0.000,C 90.000,E1 78.173} C_DIS
LIN {X 0.116,Y -359.897,Z 1284.425,A 0.000,B 0.000,C 90.000,E1 76.408} C_DIS
LIN {X 0.007,Y -349.994,Z 1284.415,A 0.000,B 0.000,C 90.000,E1 74.629} C_DIS
LIN {X 0.052,Y -338.420,Z 1284.403,A 0.000,B 0.000,C 90.000,E1 72.489} C_DIS
LIN {X -0.031,Y -323.883,Z 1284.387,A 0.000,B 0.000,C 90.000,E1 69.699} C_DIS
LIN {X -0.030,Y -307.207,Z 1284.368,A 0.000,B 0.000,C 90.000,E1 66.177} C_DIS
LIN {X -0.092,Y -296.195,Z 1284.353,A 0.000,B 0.000,C 90.000,E1 63.563} C_DIS
LIN {X 0.128,Y -287.626,Z 1284.340,A 0.000,B 0.000,C 90.000,E1 61.179} C_DIS
LIN {X 0.116,Y -277.857,Z 1284.323,A 0.000,B 0.000,C 90.000,E1 58.122} C_DIS
LIN {X -0.010,Y -268.043,Z 1284.304,A 0.000,B 0.000,C 90.000,E1 54.689} C_DIS
LIN {X -0.142,Y -260.715,Z 1284.288,A 0.000,B 0.000,C 90.000,E1 51.904} C_DIS
LIN {X 0.023,Y -253.655,Z 1284.272,A 0.000,B 0.000,C 90.000,E1 49.013} C_DIS
LIN {X -0.039,Y -246.850,Z 1284.256,A 0.000,B 0.000,C 90.000,E1 46.134} C_DIS
LIN {X 0.026,Y -238.792,Z 1284.236,A 0.000,B 0.000,C 90.000,E1 42.447} C_DIS
LIN {X -0.110,Y -231.380,Z 1284.215,A 0.000,B 0.000,C 90.000,E1 38.749} C_DIS
LIN {X -0.038,Y -224.854,Z 1284.194,A 0.000,B 0.000,C 90.000,E1 34.945} C_DIS
LIN {X -0.126,Y -219.064,Z 1284.173,A 0.000,B 0.000,C 90.000,E1 31.131} C_DIS
LIN {X 0.033,Y -214.003,Z 1284.151,A 0.000,B 0.000,C 90.000,E1 27.206} C_DIS
LIN {X 0.115,Y -209.497,Z 1284.129,A 0.000,B 0.000,C 90.000,E1 23.259} C_DIS
LIN {X 0.022,Y -205.591,Z 1284.107,A 0.000,B 0.000,C 90.000,E1 19.322} C_DIS
LIN {X -0.018,Y -201.554,Z 1284.081,A 0.000,B 0.000,C 90.000,E1 14.537} C_DIS
LIN {X 0.089,Y -198.113,Z 1284.049,A 0.000,B 0.000,C 90.000,E1 8.859} C_DIS
LIN {X 0.043,Y -195.744,Z 1284.004,A 0.000,B 0.000,C 90.000,E1 0.745} C_DIS
LIN {X 0.029,Y -197.416,Z 1283.952,A 0.000,B 0.000,C 90.000,E1 351.376} C_DIS
LIN {X 0.038,Y -200.886,Z 1283.921,A 0.000,B 0.000,C 90.000,E1 345.700} C_DIS
LIN {X -0.099,Y -205.019,Z 1283.894,A 0.000,B 0.000,C 90.000,E1 340.913} C_DIS
LIN {X -0.083,Y -209.258,Z 1283.872,A 0.000,B 0.000,C 90.000,E1 336.922} C_DIS
LIN {X 0.008,Y -214.240,Z 1283.850,A 0.000,B 0.000,C 90.000,E1 332.948} C_DIS
LIN {X -0.117,Y -219.948,Z 1283.828,A 0.000,B 0.000,C 90.000,E1 329.076} C_DIS
LIN {X 0.024,Y -226.501,Z 1283.807,A 0.000,B 0.000,C 90.000,E1 325.182} C_DIS
LIN {X 0.035,Y -233.950,Z 1283.786,A 0.000,B 0.000,C 90.000,E1 321.376} C_DIS
LIN {X 0.027,Y -242.332,Z 1283.765,A 0.000,B 0.000,C 90.000,E1 317.634} C_DIS
LIN {X -0.112,Y -250.928,Z 1283.746,A 0.000,B 0.000,C 90.000,E1 314.352} C_DIS
LIN {X -0.045,Y -257.283,Z 1283.734,A 0.000,B 0.000,C 90.000,E1 312.162} C_DIS
LIN {X -0.025,Y -264.469,Z 1283.722,A 0.000,B 0.000,C 90.000,E1 310.011} C_DIS
LIN {X -0.082,Y -271.129,Z 1283.712,A 0.000,B 0.000,C 90.000,E1 308.257} C_DIS
LIN {X -0.095,Y -280.040,Z 1283.701,A 0.000,B 0.000,C 90.000,E1 306.171} C_DIS
LIN {X -0.107,Y -290.012,Z 1283.689,A 0.000,B 0.000,C 90.000,E1 304.119} C_DIS
LIN {X -0.007,Y -301.087,Z 1283.678,A 0.000,B 0.000,C 90.000,E1 302.084} C_DIS
LIN {X -0.148,Y -311.423,Z 1283.669,A 0.000,B 0.000,C 90.000,E1 300.463} C_DIS
LIN {X -0.006,Y -327.720,Z 1283.656,A 0.000,B 0.000,C 90.000,E1 298.180} C_DIS
LIN {X 0.072,Y -347.932,Z 1283.643,A 0.000,B 0.000,C 90.000,E1 295.668} C_DIS
LIN {X -0.078,Y -363.448,Z 1283.633,A 0.000,B 0.000,C 90.000,E1 293.898} C_DIS
LIN {X 0.058,Y -376.220,Z 1283.625,A 0.000,B 0.000,C 90.000,E1 292.408} C_DIS
LIN {X 0.026,Y -388.548,Z 1283.617,A 0.000,B 0.000,C 90.000,E1 290.972} C_DIS
LIN {X -0.035,Y -413.505,Z 1283.601,A 0.000,B 0.000,C 90.000,E1 288.181} C_DIS
LIN {X -0.041,Y -423.386,Z 1283.595,A 0.000,B 0.000,C 90.000,E1 287.094} C_DIS
LIN {X 0.118,Y -430.456,Z 1283.590,A 0.000,B 0.000,C 90.000,E1 286.260} C_DIS
LIN {X -0.080,Y -437.058,Z 1283.586,A 0.000,B 0.000,C 90.000,E1 285.481} C_DIS
LIN {X 0.095,Y -443.014,Z 1283.582,A 0.000,B 0.000,C 90.000,E1 284.662} C_DIS
LIN {X 0.002,Y -448.289,Z 1283.577,A 0.000,B 0.000,C 90.000,E1 283.883} C_DIS
LIN {X -0.151,Y -452.871,Z 1283.573,A 0.000,B 0.000,C 90.000,E1 283.119} C_DIS
LIN {X 0.176,Y -456.812,Z 1283.568,A 0.000,B 0.000,C 90.000,E1 282.299} C_DIS
LIN {X -0.179,Y -459.100,Z 1283.566,A 0.000,B 0.000,C 90.000,E1 281.827} C_DIS
LIN {X -0.074,Y -461.112,Z 1283.563,A 0.000,B 0.000,C 90.000,E1 281.299} C_DIS
LIN {X -0.051,Y -462.819,Z 1283.560,A 0.000,B 0.000,C 90.000,E1 280.782} C_DIS
LIN {X 0.074,Y -464.207,Z 1283.557,A 0.000,B 0.000,C 90.000,E1 280.254} C_DIS
LIN {X 0.206,Y -465.286,Z 1283.554,A 0.000,B 0.000,C 90.000,E1 279.726} C_DIS
LIN {X -0.192,Y -465.962,Z 1283.551,A 0.000,B 0.000,C 90.000,E1 279.265} C_DIS
LIN {X -0.122,Y -466.266,Z 1283.548,A 0.000,B 0.000,C 90.000,E1 278.746} C_DIS
LIN {X 0.023,Y -466.140,Z 1283.546,A 0.000,B 0.000,C 90.000,E1 278.219} C_DIS
LIN {X 0.101,Y -465.608,Z 1283.543,A 0.000,B 0.000,C 90.000,E1 277.701} C_DIS
LIN {X 0.179,Y -464.537,Z 1283.540,A 0.000,B 0.000,C 90.000,E1 277.182} C_DIS
LIN {X -0.205,Y -463.045,Z 1283.537,A 0.000,B 0.000,C 90.000,E1 276.720} C_DIS
LIN {X 0.150,Y -459.936,Z 1283.533,A 0.000,B 0.000,C 90.000,E1 275.910} C_DIS
LIN {X 0.199,Y -457.512,Z 1283.530,A 0.000,B 0.000,C 90.000,E1 275.391} C_DIS
LIN {X 0.191,Y -454.622,Z 1283.527,A 0.000,B 0.000,C 90.000,E1 274.878} C_DIS
LIN {X 0.209,Y -451.179,Z 1283.524,A 0.000,B 0.000,C 90.000,E1 274.359} C_DIS
LIN {X 0.206,Y -446.817,Z 1283.521,A 0.000,B 0.000,C 90.000,E1 273.841} C_DIS
LIN {X -0.212,Y -441.401,Z 1283.519,A 0.000,B 0.000,C 90.000,E1 273.383} C_DIS
LIN {X 0.160,Y -435.263,Z 1283.516,A 0.000,B 0.000,C 90.000,E1 272.865} C_DIS
LIN {X 0.132,Y -428.771,Z 1283.514,A 0.000,B 0.000,C 90.000,E1 272.465} C_DIS
LIN {X 0.143,Y -421.967,Z 1283.512,A 0.000,B 0.000,C 90.000,E1 272.121} C_DIS
LIN {X 0.146,Y -414.950,Z 1283.510,A 0.000,B 0.000,C 90.000,E1 271.835} C_DIS
LIN {X 0.091,Y -407.840,Z 1283.509,A 0.000,B 0.000,C 90.000,E1 271.604} C_DIS
LIN {X -0.115,Y -400.821,Z 1283.508,A 0.000,B 0.000,C 90.000,E1 271.432} C_DIS
LIN {X -0.101,Y -393.449,Z 1283.507,A 0.000,B 0.000,C 90.000,E1 271.260} C_DIS
LIN {X 0.139,Y -385.350,Z 1283.506,A 0.000,B 0.000,C 90.000,E1 271.088} C_DIS
LIN {X -0.179,Y -376.241,Z 1283.506,A 0.000,B 0.000,C 90.000,E1 271.031} C_DIS
LIN {X 0.039,Y -363.589,Z 1283.505,A 0.000,B 0.000,C 90.000,E1 270.917} C_DIS
LIN {X -0.018,Y -355.850,Z 1283.505,A 0.000,B 0.000,C 90.000,E1 270.917} C_DIS
LIN {X -0.037,Y -181.478,Z 1283.505,A 0.000,B 0.000,C 90.000,E1 270.917} C_DIS
LIN {X -0.018,Y -181.537,Z 1283.499,A 0.000,B 0.000,C 90.000,E1 269.885} C_DIS
LIN {X -0.075,Y -180.907,Z 1283.475,A 0.000,B 0.000,C 90.000,E1 265.527} C_DIS
LIN {X -0.018,Y -180.751,Z 1283.470,A 0.000,B 0.000,C 90.000,E1 264.666} C_DIS
LIN {X 0.051,Y -178.843,Z 1283.442,A 0.000,B 0.000,C 90.000,E1 259.577} C_DIS
LIN {X -0.053,Y -175.887,Z 1283.414,A 0.000,B 0.000,C 90.000,E1 254.519} C_DIS
LIN {X 0.053,Y -174.554,Z 1283.404,A 0.000,B 0.000,C 90.000,E1 252.779} C_DIS
LIN {X -0.078,Y -171.539,Z 1283.381,A 0.000,B 0.000,C 90.000,E1 248.539} C_DIS
LIN {X -0.021,Y -167.763,Z 1283.357,A 0.000,B 0.000,C 90.000,E1 244.204} C_DIS
LIN {X -0.079,Y -166.470,Z 1283.347,A 0.000,B 0.000,C 90.000,E1 242.487} C_DIS
LIN {X 0.057,Y -163.184,Z 1283.328,A 0.000,B 0.000,C 90.000,E1 238.948} C_DIS
LIN {X -0.028,Y -161.145,Z 1283.313,A 0.000,B 0.000,C 90.000,E1 236.342} C_DIS
LIN {X 0.008,Y -157.164,Z 1283.288,A 0.000,B 0.000,C 90.000,E1 231.904} C_DIS
LIN {X 0.031,Y -155.896,Z 1283.278,A 0.000,B 0.000,C 90.000,E1 230.114} C_DIS
LIN {X -0.011,Y -152.146,Z 1283.254,A 0.000,B 0.000,C 90.000,E1 225.648} C_DIS
LIN {X 0.009,Y -150.395,Z 1283.239,A 0.000,B 0.000,C 90.000,E1 222.933} C_DIS
LIN {X 0.033,Y -147.126,Z 1283.213,A 0.000,B 0.000,C 90.000,E1 218.382} C_DIS
LIN {X 0.023,Y -145.689,Z 1283.198,A 0.000,B 0.000,C 90.000,E1 215.644} C_DIS
LIN {X 0.021,Y -143.071,Z 1283.173,A 0.000,B 0.000,C 90.000,E1 211.052} C_DIS
LIN {X -0.048,Y -141.692,Z 1283.152,A 0.000,B 0.000,C 90.000,E1 207.385} C_DIS
LIN {X 0.007,Y -139.462,Z 1283.116,A 0.000,B 0.000,C 90.000,E1 200.865} C_DIS
LIN {X -0.070,Y -139.195,Z 1283.106,A 0.000,B 0.000,C 90.000,E1 199.033} C_DIS
LIN {X -0.007,Y -138.325,Z 1283.054,A 0.000,B 0.000,C 90.000,E1 189.670} C_DIS
LIN {X -0.002,Y -139.450,Z 1283.007,A 0.000,B 0.000,C 90.000,E1 181.260} C_DIS
LIN {X -0.062,Y -140.994,Z 1282.976,A 0.000,B 0.000,C 90.000,E1 175.698} C_DIS
LIN {X 0.029,Y -142.748,Z 1282.955,A 0.000,B 0.000,C 90.000,E1 171.951} C_DIS
LIN {X -0.015,Y -145.147,Z 1282.930,A 0.000,B 0.000,C 90.000,E1 167.353} C_DIS
LIN {X -0.022,Y -147.770,Z 1282.909,A 0.000,B 0.000,C 90.000,E1 163.685} C_DIS
LIN {X 0.058,Y -150.444,Z 1282.889,A 0.000,B 0.000,C 90.000,E1 160.007} C_DIS
LIN {X -0.008,Y -153.891,Z 1282.869,A 0.000,B 0.000,C 90.000,E1 156.410} C_DIS
LIN {X -0.014,Y -157.301,Z 1282.849,A 0.000,B 0.000,C 90.000,E1 152.820} C_DIS
LIN {X 0.005,Y -161.486,Z 1282.829,A 0.000,B 0.000,C 90.000,E1 149.253} C_DIS
LIN {X 0.021,Y -165.684,Z 1282.810,A 0.000,B 0.000,C 90.000,E1 145.722} C_DIS
LIN {X -0.092,Y -170.626,Z 1282.790,A 0.000,B 0.000,C 90.000,E1 142.271} C_DIS
LIN {X 0.062,Y -175.503,Z 1282.771,A 0.000,B 0.000,C 90.000,E1 138.771} C_DIS
LIN {X -0.072,Y -181.123,Z 1282.752,A 0.000,B 0.000,C 90.000,E1 135.405} C_DIS
LIN {X 0.054,Y -186.571,Z 1282.733,A 0.000,B 0.000,C 90.000,E1 132.000} C_DIS
LIN {X 0.004,Y -191.184,Z 1282.720,A 0.000,B 0.000,C 90.000,E1 129.519} C_DIS
LIN {X 0.050,Y -196.992,Z 1282.701,A 0.000,B 0.000,C 90.000,E1 126.217} C_DIS
LIN {X -0.014,Y -199.820,Z 1282.693,A 0.000,B 0.000,C 90.000,E1 124.818} C_DIS
LIN {X -0.058,Y -309.140,Z 1282.693,A 0.000,B 0.000,C 90.000,E1 124.818} C_DIS
LIN {X -0.049,Y -315.227,Z 1282.692,A 0.000,B 0.000,C 90.000,E1 124.612} C_DIS
LIN {X -0.078,Y -317.930,Z 1282.691,A 0.000,B 0.000,C 90.000,E1 124.405} C_DIS
LIN {X 0.107,Y -321.704,Z 1282.688,A 0.000,B 0.000,C 90.000,E1 123.913} C_DIS
LIN {X -0.087,Y -323.526,Z 1282.687,A 0.000,B 0.000,C 90.000,E1 123.627} C_DIS
LIN {X -0.012,Y -324.943,Z 1282.685,A 0.000,B 0.000,C 90.000,E1 123.293} C_DIS
LIN {X 0.083,Y -336.641,Z 1282.667,A 0.000,B 0.000,C 90.000,E1 120.129} C_DIS
LIN {X -0.121,Y -348.559,Z 1282.652,A 0.000,B 0.000,C 90.000,E1 117.385} C_DIS
LIN {X 0.000,Y -361.936,Z 1282.637,A 0.000,B 0.000,C 90.000,E1 114.643} C_DIS
LIN {X -0.036,Y -375.143,Z 1282.624,A 0.000,B 0.000,C 90.000,E1 112.280} C_DIS
LIN {X 0.123,Y -389.684,Z 1282.611,A 0.000,B 0.000,C 90.000,E1 109.939} C_DIS
LIN {X 0.003,Y -405.664,Z 1282.598,A 0.000,B 0.000,C 90.000,E1 107.692} C_DIS
LIN {X 0.021,Y -423.192,Z 1282.586,A 0.000,B 0.000,C 90.000,E1 105.481} C_DIS
LIN {X -0.143,Y -442.363,Z 1282.574,A 0.000,B 0.000,C 90.000,E1 103.355} C_DIS
LIN {X 0.265,Y -462.467,Z 1282.563,A 0.000,B 0.000,C 90.000,E1 101.299} C_DIS
LIN {X 0.187,Y -475.296,Z 1282.557,A 0.000,B 0.000,C 90.000,E1 100.141} C_DIS
LIN {X -0.216,Y -477.579,Z 1282.555,A 0.000,B 0.000,C 90.000,E1 99.962} C_DIS
LIN {X 0.170,Y -479.417,Z 1282.554,A 0.000,B 0.000,C 90.000,E1 99.670} C_DIS
LIN {X 0.006,Y -480.805,Z 1282.552,A 0.000,B 0.000,C 90.000,E1 99.443} C_DIS
LIN {X 0.239,Y -482.605,Z 1282.550,A 0.000,B 0.000,C 90.000,E1 98.916} C_DIS
LIN {X -0.075,Y -483.307,Z 1282.547,A 0.000,B 0.000,C 90.000,E1 98.454} C_DIS
LIN {X 0.103,Y -483.029,Z 1282.544,A 0.000,B 0.000,C 90.000,E1 97.936} C_DIS
LIN {X -0.130,Y -481.731,Z 1282.541,A 0.000,B 0.000,C 90.000,E1 97.466} C_DIS
LIN {X 0.168,Y -480.635,Z 1282.540,A 0.000,B 0.000,C 90.000,E1 97.182} C_DIS
LIN {X 0.048,Y -479.166,Z 1282.539,A 0.000,B 0.000,C 90.000,E1 96.947} C_DIS
LIN {X -0.113,Y -462.601,Z 1282.526,A 0.000,B 0.000,C 90.000,E1 94.702} C_DIS
LIN {X -0.077,Y -445.328,Z 1282.512,A 0.000,B 0.000,C 90.000,E1 92.121} C_DIS
LIN {X 0.032,Y -432.443,Z 1282.500,A 0.000,B 0.000,C 90.000,E1 90.000} C_DIS
LIN {X 0.073,Y -417.699,Z 1282.485,A 0.000,B 0.000,C 90.000,E1 87.306} C_DIS
LIN {X 0.011,Y -406.106,Z 1282.473,A 0.000,B 0.000,C 90.000,E1 85.122} C_DIS
LIN {X 0.022,Y -397.423,Z 1282.464,A 0.000,B 0.000,C 90.000,E1 83.451} C_DIS
LIN {X -0.128,Y -388.583,Z 1282.454,A 0.000,B 0.000,C 90.000,E1 81.781} C_DIS
LIN {X 0.053,Y -379.520,Z 1282.445,A 0.000,B 0.000,C 90.000,E1 80.038} C_DIS
LIN {X 0.134,Y -371.714,Z 1282.437,A 0.000,B 0.000,C 90.000,E1 78.578} C_DIS
LIN {X 0.070,Y -362.009,Z 1282.427,A 0.000,B 0.000,C 90.000,E1 76.825} C_DIS
LIN {X -0.003,Y -352.111,Z 1282.417,A 0.000,B 0.000,C 90.000,E1 75.046} C_DIS
LIN {X 0.084,Y -340.534,Z 1282.405,A 0.000,B 0.000,C 90.000,E1 72.906} C_DIS
LIN {X 0.093,Y -327.539,Z 1282.391,A 0.000,B 0.000,C 90.000,E1 70.423} C_DIS
LIN {X 0.097,Y -310.596,Z 1282.372,A 0.000,B 0.000,C 90.000,E1 66.922} C_DIS
LIN {X -0.134,Y -297.940,Z 1282.356,A 0.000,B 0.000,C 90.000,E1 64.024} C_DIS
LIN {X -0.121,Y -290.358,Z 1282.344,A 0.000,B 0.000,C 90.000,E1 62.025} C_DIS
LIN {X 0.035,Y -280.250,Z 1282.328,A 0.000,B 0.000,C 90.000,E1 58.948} C_DIS
LIN {X -0.021,Y -270.176,Z 1282.308,A 0.000,B 0.000,C 90.000,E1 55.515} C_DIS
LIN {X 0.076,Y -260.894,Z 1282.289,A 0.000,B 0.000,C 90.000,E1 51.984} C_DIS
LIN {X 0.046,Y -253.803,Z 1282.273,A 0.000,B 0.000,C 90.000,E1 49.138} C_DIS
LIN {X -0.006,Y -246.975,Z 1282.257,A 0.000,B 0.000,C 90.000,E1 46.257} C_DIS
LIN {X -0.103,Y -238.917,Z 1282.237,A 0.000,B 0.000,C 90.000,E1 42.609} C_DIS
LIN {X 0.098,Y -231.466,Z 1282.216,A 0.000,B 0.000,C 90.000,E1 38.830} C_DIS
LIN {X -0.144,Y -224.876,Z 1282.195,A 0.000,B 0.000,C 90.000,E1 35.105} C_DIS
LIN {X 0.081,Y -219.031,Z 1282.173,A 0.000,B 0.000,C 90.000,E1 31.209} C_DIS
LIN {X 0.047,Y -213.877,Z 1282.152,A 0.000,B 0.000,C 90.000,E1 27.334} C_DIS
LIN {X 0.126,Y -209.292,Z 1282.130,A 0.000,B 0.000,C 90.000,E1 23.387} C_DIS
LIN {X 0.029,Y -205.362,Z 1282.108,A 0.000,B 0.000,C 90.000,E1 19.450} C_DIS
LIN {X -0.013,Y -201.299,Z 1282.081,A 0.000,B 0.000,C 90.000,E1 14.662} C_DIS
LIN {X -0.071,Y -197.837,Z 1282.050,A 0.000,B 0.000,C 90.000,E1 9.029} C_DIS
LIN {X 0.054,Y -195.473,Z 1282.005,A 0.000,B 0.000,C 90.000,E1 0.859} C_DIS
LIN {X 0.014,Y -197.261,Z 1281.952,A 0.000,B 0.000,C 90.000,E1 351.376} C_DIS
LIN {X 0.017,Y -200.792,Z 1281.921,A 0.000,B 0.000,C 90.000,E1 345.700} C_DIS
LIN {X 0.071,Y -204.969,Z 1281.894,A 0.000,B 0.000,C 90.000,E1 340.859} C_DIS
LIN {X -0.110,Y -209.234,Z 1281.872,A 0.000,B 0.000,C 90.000,E1 336.922} C_DIS
LIN {X -0.019,Y -214.233,Z 1281.850,A 0.000,B 0.000,C 90.000,E1 332.948} C_DIS
LIN {X -0.145,Y -219.956,Z 1281.828,A 0.000,B 0.000,C 90.000,E1 329.076} C_DIS
LIN {X -0.005,Y -226.533,Z 1281.807,A 0.000,B 0.000,C 90.000,E1 325.182} C_DIS
LIN {X 0.005,Y -233.988,Z 1281.785,A 0.000,B 0.000,C 90.000,E1 321.376} C_DIS
LIN {X -0.001,Y -242.354,Z 1281.765,A 0.000,B 0.000,C 90.000,E1 317.634} C_DIS
LIN {X 0.038,Y -249.935,Z 1281.748,A 0.000,B 0.000,C 90.000,E1 314.676} C_DIS
LIN {X -0.076,Y -257.271,Z 1281.734,A 0.000,B 0.000,C 90.000,E1 312.162} C_DIS
LIN {X -0.056,Y -264.437,Z 1281.722,A 0.000,B 0.000,C 90.000,E1 310.011} C_DIS
LIN {X 0.054,Y -271.092,Z 1281.712,A 0.000,B 0.000,C 90.000,E1 308.222} C_DIS
LIN {X 0.035,Y -280.012,Z 1281.701,A 0.000,B 0.000,C 90.000,E1 306.137} C_DIS
LIN {X -0.143,Y -289.991,Z 1281.689,A 0.000,B 0.000,C 90.000,E1 304.119} C_DIS
LIN {X -0.045,Y -301.049,Z 1281.678,A 0.000,B 0.000,C 90.000,E1 302.084} C_DIS
LIN {X 0.081,Y -311.357,Z 1281.669,A 0.000,B 0.000,C 90.000,E1 300.413} C_DIS
LIN {X 0.105,Y -327.660,Z 1281.656,A 0.000,B 0.000,C 90.000,E1 298.153} C_DIS
LIN {X 0.038,Y -347.847,Z 1281.643,A 0.000,B 0.000,C 90.000,E1 295.668} C_DIS
LIN {X -0.158,Y -363.437,Z 1281.633,A 0.000,B 0.000,C 90.000,E1 293.898} C_DIS
LIN {X 0.076,Y -376.273,Z 1281.624,A 0.000,B 0.000,C 90.000,E1 292.386} C_DIS
LIN {X 0.123,Y -386.185,Z 1281.618,A 0.000,B 0.000,C 90.000,E1 291.227} C_DIS
LIN {X 0.177,Y -410.987,Z 1281.602,A 0.000,B 0.000,C 90.000,E1 288.417} C_DIS
LIN {X -0.080,Y -418.563,Z 1281.598,A 0.000,B 0.000,C 90.000,E1 287.638} C_DIS
LIN {X -0.109,Y -428.233,Z 1281.592,A 0.000,B 0.000,C 90.000,E1 286.551} C_DIS
LIN {X 0.094,Y -434.986,Z 1281.587,A 0.000,B 0.000,C 90.000,E1 285.717} C_DIS
LIN {X -0.183,Y -441.203,Z 1281.583,A 0.000,B 0.000,C 90.000,E1 284.954} C_DIS
LIN {X 0.143,Y -446.675,Z 1281.578,A 0.000,B 0.000,C 90.000,E1 284.120} C_DIS
LIN {X -0.027,Y -451.526,Z 1281.574,A 0.000,B 0.000,C 90.000,E1 283.355} C_DIS
LIN {X -0.152,Y -455.727,Z 1281.570,A 0.000,B 0.000,C 90.000,E1 282.591} C_DIS
LIN {X 0.204,Y -459.217,Z 1281.566,A 0.000,B 0.000,C 90.000,E1 281.771} C_DIS
LIN {X -0.140,Y -461.192,Z 1281.563,A 0.000,B 0.000,C 90.000,E1 281.299} C_DIS
LIN {X -0.116,Y -462.916,Z 1281.560,A 0.000,B 0.000,C 90.000,E1 280.782} C_DIS
LIN {X 0.008,Y -464.322,Z 1281.557,A 0.000,B 0.000,C 90.000,E1 280.254} C_DIS
LIN {X 0.141,Y -465.365,Z 1281.554,A 0.000,B 0.000,C 90.000,E1 279.726} C_DIS
LIN {X 0.204,Y -466.053,Z 1281.551,A 0.000,B 0.000,C 90.000,E1 279.208} C_DIS
LIN {X -0.185,Y -466.391,Z 1281.548,A 0.000,B 0.000,C 90.000,E1 278.746} C_DIS
LIN {X -0.041,Y -466.263,Z 1281.546,A 0.000,B 0.000,C 90.000,E1 278.219} C_DIS
LIN {X 0.038,Y -465.721,Z 1281.543,A 0.000,B 0.000,C 90.000,E1 277.701} C_DIS
LIN {X 0.118,Y -464.695,Z 1281.540,A 0.000,B 0.000,C 90.000,E1 277.182} C_DIS
LIN {X 0.195,Y -463.198,Z 1281.537,A 0.000,B 0.000,C 90.000,E1 276.663} C_DIS
LIN {X 0.090,Y -460.157,Z 1281.533,A 0.000,B 0.000,C 90.000,E1 275.910} C_DIS
LIN {X -0.087,Y -456.430,Z 1281.529,A 0.000,B 0.000,C 90.000,E1 275.163} C_DIS
LIN {X -0.058,Y -453.351,Z 1281.526,A 0.000,B 0.000,C 90.000,E1 274.645} C_DIS
LIN {X -0.080,Y -449.503,Z 1281.523,A 0.000,B 0.000,C 90.000,E1 274.131} C_DIS
LIN {X 0.155,Y -447.257,Z 1281.521,A 0.000,B 0.000,C 90.000,E1 273.841} C_DIS
LIN {X 0.156,Y -441.870,Z 1281.519,A 0.000,B 0.000,C 90.000,E1 273.326} C_DIS
LIN {X 0.049,Y -435.713,Z 1281.516,A 0.000,B 0.000,C 90.000,E1 272.865} C_DIS
